Yaskawa INFORM job: OK_R2_O8B-O21B(90,0)_KMOK_HARDOX.JBI

/JOB
//NAME OK_R2_O8B-O21B(90,0)_KMOK_HARDOX
///FOLDERNAME X4
//POS
///NPOS 686,686,686,29,0,0
///TOOL 0
///POSTYPE PULSE
///PULSE
C00000=-91699,-114837,-126172,5297,65572,69852
C00001=-92194,-112793,-113721,5907,59024,69345
C00002=-143897,-89142,-104886,30363,76848,53183
C00003=-141756,-87617,-100734,29753,74573,53385
C00004=-141756,-87858,-100091,29820,74119,53263
C00005=-141756,-87802,-100249,29804,74230,53293
C00006=-141244,-84255,-98746,29497,74846,53651
C00007=-141653,-86886,-101326,29626,75189,53586
C00008=-110766,-103587,-109768,16030,63754,62789
C00009=-110766,-104046,-107477,16255,62170,62558
C00010=-110766,-104165,-106515,16351,61543,62463
C00011=-110766,-104147,-106683,16334,61651,62479
C00012=-111036,-99665,-105018,16294,62933,62564
C00013=-110753,-104252,-107692,16244,62194,62563
C00014=-67116,-81864,-100907,-8307,67410,78303
C00015=-67696,-81353,-98479,-8065,66136,78195
C00016=-67696,-81727,-97702,-8106,65471,78242
C00017=-67696,-81654,-97861,-8098,65606,78232
C00018=-68924,-78441,-96430,-7380,66259,77758
C00019=-67562,-81507,-99004,-8124,66390,78224
C00020=-94591,-107711,-114910,7081,62535,68652
C00021=-75177,-96078,-118139,30635,103857,-57240
C00022=-71016,-101172,-117038,29652,99603,-56842
C00023=-69320,-102842,-116458,29300,97976,-56637
C00024=-65815,-114376,-118551,28520,92729,-56653
C00025=-65815,-114603,-117718,28482,92175,-56787
C00026=-65333,-115185,-120736,28492,93393,-56311
C00027=-69320,-102842,-116458,29300,97976,-56637
C00028=-95175,-93300,-89498,59989,102155,-86131
C00029=-94783,-95327,-90301,59871,101628,-86283
C00030=-95175,-93300,-89498,59989,102155,-86131
C00031=-95403,-90904,-93442,60883,104178,-84663
C00032=-96846,-88575,-93381,61258,105655,-84430
C00033=-100267,-82342,-92970,62384,109223,-83757
C00034=-98853,-105972,-123361,35115,85568,-62201
C00035=-123874,-116503,-132949,35316,93358,-57662
C00036=-98784,-130821,-129289,12660,72810,-27269
C00037=-95442,-119682,-123188,11300,74256,-25961
C00038=-89918,-115832,-119261,9213,73142,-24151
C00039=-89918,-116068,-118310,9245,72445,-24204
C00040=-89918,-115832,-119261,9213,73142,-24151
C00041=-86534,-112000,-117975,7848,73961,-22933
C00042=-89918,-115832,-119261,9213,73142,-24151
C00043=-91545,-105966,-115876,9715,76271,-24462
C00044=-89918,-115832,-119261,9213,73142,-24151
C00045=-100559,-101270,-121421,12879,83175,-26784
C00046=-103898,-109015,-126857,14089,83070,-27872
C00047=-112603,-104533,-117877,29713,115926,-66306
C00048=-112603,-104533,-117877,29713,115926,-66306
C00049=-102787,-102282,-117268,28859,121596,-74546
C00050=-102787,-103288,-115881,28417,120387,-74903
C00051=-102787,-102191,-117377,28898,121696,-74514
C00052=-102247,-107992,-119426,28435,120002,-74778
C00053=-104853,-110239,-121572,27980,116786,-76632
C00054=-123177,-144145,-129947,26642,102859,-76425
C00055=-123829,-162749,-132848,26863,92935,-75206
C00056=-121638,-162916,-132889,27033,92171,-74551
C00057=-123829,-165003,-135169,26874,93176,-75150
C00058=-112500,-101779,-108680,28673,112161,-67324
C00059=-131997,-56357,-109229,-4920,90907,-66095
C00060=-147842,-82951,-112210,-34984,98309,-69155
C00061=-149737,-87239,-109966,-34223,94635,-68708
C00062=-151378,-90687,-107740,-33690,91394,-68340
C00063=-151378,-91074,-107136,-33673,90915,-68196
C00064=-151378,-90687,-107740,-33690,91394,-68340
C00065=-145558,-100693,-110774,-34812,90892,-65938
C00066=-145748,-102567,-109629,-34742,89434,-65557
C00067=-146398,-106855,-111180,-34614,88141,-65411
C00068=-145748,-102567,-109629,-34742,89434,-65557
C00069=-144942,-96836,-108242,-34942,91483,-65883
C00070=-124830,-105124,-96789,-55472,88700,-57654
C00071=-126521,-104925,-96716,-55344,87736,-58010
C00072=-123249,-105523,-98221,-55595,90026,-57599
C00073=-144949,-101354,-110618,-34915,90771,-65662
C00074=-150499,-88658,-108954,-33966,93222,-68562
C00075=-149737,-87239,-109966,-34223,94635,-68708
C00076=-147842,-82951,-112210,-34984,98309,-69155
C00077=-134744,-82461,-113999,-23220,99839,-19223
C00078=-107178,-113461,-99894,-5964,101445,70182
C00079=-116777,-120475,-92303,-7084,92443,67341
C00080=-117649,-121004,-89231,-7177,90217,67172
C00081=-117541,-124461,-90223,-7160,89070,67274
C00082=-117649,-121004,-89231,-7177,90217,67172
C00083=-121247,-121045,-89244,-7619,89875,65972
C00084=-117649,-121004,-89231,-7177,90217,67172
C00085=-120454,-123758,-93756,-7530,91322,66155
C00086=-131821,-147240,-100571,-7170,74455,63187
C00087=-132564,-146887,-99168,-7097,73320,62988
C00088=-132564,-147261,-99594,-7095,73390,62984
C00089=-116129,-123152,-95240,-7006,92928,67534
C00090=-114019,-118624,-94636,-6761,95050,68140
C00091=-115483,-77500,-114184,15325,109930,22258
C00092=-107117,-124945,-135933,-21570,97656,8797
C00093=-118143,-111392,-129277,-15030,88270,-9704
C00094=-118164,-109444,-128626,-15025,88847,-9780
C00095=-118164,-110450,-128026,-15024,87989,-9675
C00096=-118164,-110074,-128260,-15024,88315,-9716
C00097=-118257,-101380,-125250,-15013,90827,-10051
C00098=-118164,-108155,-129289,-15031,89881,-9907
C00099=-110085,-126828,-135239,-17345,85673,-6704
C00100=-92891,-111374,-130366,-26323,94899,34453
C00101=-97190,-111538,-124535,-25207,90331,33950
C00102=-98877,-113015,-125031,-24804,89436,33545
C00103=-97190,-111538,-124535,-25207,90331,33950
C00104=-97263,-106439,-128356,-25089,94874,32878
C00105=-81189,-95371,-128319,620,93628,-17487
C00106=-93710,-100817,-120600,-17770,81443,-35553
C00107=-93248,-94915,-114871,-17964,81066,-35345
C00108=-93496,-90946,-110472,-17900,80379,-35326
C00109=-93496,-91762,-109449,-17950,79378,-35179
C00110=-93496,-91644,-109606,-17943,79529,-35199
C00111=-94018,-88323,-108262,-17704,80263,-35482
C00112=-93496,-90946,-110472,-17900,80379,-35326
C00113=-94462,-94397,-113311,-17534,80159,-35616
C00114=-94975,-100261,-119034,-17317,80544,-35841
C00115=-122852,-136172,-128581,30503,68555,23673
C00116=-143305,-96642,-110194,35986,83923,20153
C00117=-143305,-96740,-110018,35993,83793,20110
C00118=-143305,-97404,-108670,36055,82835,19796
C00119=-143221,-96691,-108564,36013,83047,19900
C00120=-142576,-91782,-106634,35760,83882,20426
C00121=-143221,-96196,-109551,35968,83751,20131
C00122=-150080,-145633,-129217,38890,75983,14564
C00123=-150642,-143359,-125500,39162,75356,14082
C00124=-150642,-142275,-123303,39286,74731,13847
C00125=-150642,-142343,-123438,39278,74769,13861
C00126=-149456,-135964,-121650,38723,75947,14827
C00127=-150182,-141675,-125924,38909,76032,14540
C00128=-92946,-121634,-121424,16744,62834,34226
C00129=-86370,-109059,-114128,13073,63567,36806
C00130=-86370,-109316,-113053,13160,62794,36714
C00131=-86334,-109454,-113302,13133,62869,36736
C00132=-87103,-105692,-111971,13415,64077,36592
C00133=-86334,-109252,-114136,13065,63471,36806
C00134=-121032,-150272,-131973,30968,63431,22949
C00135=-105037,-121499,-124352,-26595,83975,43332
C00136=-119038,-120466,-118045,-23113,76809,39715
C00137=-125137,-115371,-113740,-21293,75158,37787
C00138=-125137,-115377,-112598,-21357,74498,37908
C00139=-125137,-115371,-113740,-21293,75158,37787
C00140=-125247,-119622,-115037,-21389,73833,26696
C00141=-125053,-112026,-112515,-21239,76079,26360
C00142=-125247,-119622,-115037,-21389,73833,26696
C00143=-117922,-113856,-115388,-23299,78742,39741
C00144=-113283,-118224,-119490,-24564,80311,41113
C00145=-130678,-94773,-121138,-18217,87222,14080
C00146=-167942,-138091,-131423,6732,80009,27343
C00147=-170575,-113227,-120751,7300,86397,26822
C00148=-169077,-108435,-117775,6935,86895,27340
C00149=-169077,-108900,-116810,6936,86070,27295
C00150=-169077,-108794,-117048,6936,86270,27307
C00151=-170304,-106542,-116256,7229,87038,26949
C00152=-168740,-106235,-118221,6850,88265,27525
C00153=-177701,-115390,-116622,14957,80027,1616
C00154=-176753,-112936,-115506,14676,80414,1989
C00155=-175630,-109912,-114469,14334,81107,2455
C00156=-177564,-114998,-116703,14910,80246,1690
C00157=-188009,-144692,-131667,17931,76513,-2502
C00158=-152038,-126618,-128978,-10588,85958,28176
C00159=-152038,-126618,-128978,-10588,85958,28176
C00160=-152439,-128268,-129478,-10504,85377,28090
C00161=-152439,-128687,-128060,-10515,84308,28182
C00162=-152439,-128634,-128276,-10513,84466,28168
C00163=-154807,-125417,-127295,-9971,85207,27314
C00164=-152439,-127687,-130796,-10495,86471,28000
C00165=-151563,-130369,-131601,-10695,85714,28356
C00166=-164160,-102502,-129441,9384,110509,-55546
C00167=-159433,-112173,-127809,8699,104125,-54469
C00168=-159433,-113313,-126887,8650,102984,-54550
C00169=-159433,-113125,-127052,8657,103179,-54535
C00170=-157389,-116461,-128145,8463,101945,-53942
C00171=-159433,-111320,-128398,8735,104915,-54410
C00172=-152229,-108849,-132490,7833,104970,-48789
C00173=-93963,-130535,-128792,24722,74568,-16491
C00174=-90353,-119281,-117601,23619,72522,-15568
C00175=-81815,-101184,-113078,14856,80893,-11838
C00176=-81815,-101805,-111815,14897,79832,-11967
C00177=-81815,-101566,-112336,14880,80261,-11914
C00178=-81691,-96656,-110485,14792,81580,-11713
C00179=-81815,-101566,-112336,14880,80261,-11914
C00180=-94368,-118351,-115092,25106,72713,-8195
C00181=-94368,-118242,-113051,25259,71623,-8437
C00182=-92475,-116697,-112544,24567,71499,-7736
C00183=-98770,-117080,-112671,26610,73310,-9747
C00184=-98093,-111583,-112853,26067,75742,-17780
C00185=-89023,-115119,-115343,23068,72843,-15005
C00186=-90353,-119281,-117601,23619,72522,-15568
C00187=-93963,-130636,-123354,25128,71472,-17166
C00188=-112708,-151913,-126980,52913,79334,40142
C00189=-108924,-145810,-121760,52599,77119,40924
C00190=-107448,-143466,-119685,52466,76232,41216
C00191=-107548,-140507,-116374,52568,75966,41003
C00192=-107448,-143466,-119685,52466,76232,41216
C00193=-124866,-69208,-71806,74049,113649,28483
C00194=-122400,-71971,-73000,73720,111742,28428
C00195=-124866,-69208,-71806,74049,113649,28483
C00196=-131136,-146090,-96201,76130,76771,21052
C00197=-127770,-141595,-95524,76231,74990,22221
C00198=-131136,-146090,-96201,76130,76771,21052
C00199=-112467,-159247,-111976,60211,61283,24397
C00200=-113297,-157006,-110103,60230,61789,24238
C00201=-113297,-157814,-110929,60188,61836,24279
C00202=-111416,-155256,-110381,59676,61201,25079
C00203=-114119,-159107,-112646,60032,62541,24296
C00204=-145608,-121761,-102949,57803,88894,23690
C00205=-146047,-120434,-101564,57803,89067,23542
C00206=-146481,-119084,-100092,57801,89215,23379
C00207=-146481,-119516,-101126,57808,89444,23539
C00208=-144820,-117039,-100336,57803,88864,24154
C00209=-147924,-121944,-103270,57808,90363,23296
C00210=-147924,-121944,-103270,57808,90363,23296
C00211=-137007,-126621,-110171,48785,83769,25153
C00212=-137007,-126054,-108752,48822,83378,24951
C00213=-137359,-125765,-109353,48816,83916,25050
C00214=-136478,-122214,-108258,48678,84217,25648
C00215=-137706,-129591,-111729,48871,83766,24798
C00216=-138625,-143143,-124865,48877,85014,24974
C00217=-98331,-144500,-124457,41780,63547,34680
C00218=-104311,-135778,-116637,47474,67333,33513
C00219=-104982,-134568,-114900,47757,67380,33183
C00220=-104982,-134679,-115131,47731,67438,33213
C00221=-102403,-135448,-115392,47202,65913,33778
C00222=-105649,-135232,-117175,47605,68461,33397
C00223=-103532,-169539,-136511,48991,63433,31812
C00224=-103532,-169539,-136511,48991,63433,31812
C00225=-27587,-68716,-104105,-32768,107246,55193
C00226=-44542,-60786,-93895,-29075,99837,51184
C00227=-48925,-61585,-92322,-27957,97276,50292
C00228=-49957,-62195,-92636,-27707,96857,50034
C00229=-49778,-62097,-92585,-27750,96927,50079
C00230=-49778,-62949,-91655,-27679,96029,50296
C00231=-46799,-62314,-93554,-28472,98262,50792
C00232=-32844,-112560,-114598,-30217,91594,57615
C00233=-34172,-119266,-116359,-29997,89069,57770
C00234=-36208,-121107,-116949,-29726,87845,57309
C00235=-35920,-120864,-116872,-29765,88013,57375
C00236=-35920,-120756,-115116,-29769,87119,57607
C00237=-34172,-119266,-116359,-29997,89069,57770
C00238=-34009,-88694,-103453,-33144,106213,64136
C00239=-48532,-32879,-74171,-34015,109897,57248
C00240=-43788,-34488,-76749,-34872,112199,58300
C00241=-48317,-118248,-127921,-15090,82411,66271
C00242=-90179,-134235,-132818,22872,80929,49314
C00243=-142804,-125519,-116198,76046,95508,7054
C00244=-120615,-97641,-119015,9375,90228,-9949
C00245=-120987,-96376,-113097,9471,87311,-10282
C00246=-120613,-99917,-116962,9368,87826,-10128
C00247=-121552,-104751,-117459,9639,85780,-10586
C00248=-110169,-106106,-116921,6405,83791,7848
C00249=-108950,-107035,-116988,5812,83203,8687
C00250=-101778,-109524,-117401,437,81208,17199
C00251=-92910,-108806,-115845,-6377,80483,27828
C00252=-91325,-110019,-114746,-6888,79315,28418
C00253=-89437,-130785,-128831,-4407,77618,27633
C00254=-146443,-63628,-115918,-3009,102570,37934
C00255=-146980,-83801,-122033,-27049,110301,76522
C00256=-150856,-97054,-121393,-25304,102734,76951
C00257=-152223,-100571,-121286,-24887,100651,76928
C00258=-148913,-93356,-120721,-25800,104620,77205
C00259=-150557,-96944,-122901,-25470,103711,76838
C00260=-148738,-112083,-124761,-25075,98193,78687
C00261=-146683,-119723,-126910,-25161,96417,79805
C00262=-143109,-114454,-128222,-25889,100648,80164
C00263=-140673,-104492,-128634,-26873,106197,79748
C00264=-120599,-130072,-117206,-45023,91037,77550
C00265=-120599,-129119,-114227,-44983,90071,77984
C00266=-124865,-150469,-117889,-44902,76314,77260
C00267=-120042,-124581,-111856,-45029,90980,77838
C00268=-119368,-131507,-114599,-44995,89976,78605
C00269=-124285,-150580,-117667,-44961,76466,77468
C00270=-119900,-149520,-114561,-45303,77705,79000
C00271=-119479,-146252,-112177,-45280,78069,79034
C00272=-120598,-127933,-111142,-44960,89143,78399
C00273=-120599,-129048,-114177,-44983,90075,77982
C00274=-81107,-101484,-115694,35475,102250,71567
C00275=-81237,-105179,-114207,34170,99607,71777
C00276=-82059,-102607,-116004,34567,101946,72190
C00277=-81374,-98102,-114013,34658,102588,72668
C00278=-80946,-104008,-116650,25534,103675,80963
C00279=-81739,-109308,-117836,24647,100784,82296
C00280=-83058,-108491,-117286,24741,101236,81911
C00281=-79384,-104922,-115530,34104,103743,72622
C00282=-80190,-85868,-119713,25334,110684,45677
C00283=-66991,-110384,-121517,5418,108134,-76364
C00284=-56399,-121526,-132511,11086,102541,-72269
C00285=-51570,-131189,-133992,11264,103193,-70513
C00286=-26251,-133049,-134514,-2928,99563,-63672
C00287=-67233,-108188,-115958,5335,105866,-76549
C00288=-66897,-113678,-118543,5308,104619,-76489
C00289=-40340,-135502,-134832,4529,99531,-76926
C00290=-39996,-126929,-132065,1999,104723,-72189
C00291=-40582,-118742,-129232,-2204,110819,-68387
C00292=-63906,-99170,-120419,5411,122707,-74964
C00293=-69620,-108722,-123406,2860,118643,-77498
C00294=-87784,-109018,-121307,623,118193,-84117
C00295=-84930,-119629,-129782,-1888,113436,-83486
C00296=-84729,-121080,-124653,20914,107476,-65948
C00297=-95444,-112372,-114390,31511,111945,-67927
C00298=-67316,-107916,-115567,-9495,105572,-72905
C00299=-66579,-114256,-118448,-9402,104190,-72540
C00300=-98021,-122686,-116586,31197,106837,-67491
C00301=-98017,-122619,-115764,31114,106429,-67606
C00302=-102197,-111658,-121490,32833,115802,-66493
C00303=-86428,-100957,-127747,22004,113840,-67454
C00304=-53800,-100419,-127772,-3487,91936,-72900
C00305=-55487,-108533,-124083,-2963,85444,-73257
C00306=-76650,-116115,-116137,28754,70174,-77169
C00307=-54376,-102036,-122875,-3303,88076,-72973
C00308=-53684,-106892,-125333,-3516,87122,-72731
C00309=-74308,-115452,-115917,27821,69577,-76396
C00310=-59122,-109220,-113787,21025,66918,-71130
C00311=-57844,-108351,-113482,20394,66848,-70662
C00312=-53834,-105518,-125265,-3470,87779,-72796
C00313=-58883,-114751,-131257,-1913,86567,-74352
C00314=-99205,-132197,-126076,29274,71590,12900
C00315=-100538,-139639,-126656,10769,67376,15479
C00316=-99890,-133434,-123018,10459,68226,15794
C00317=-121557,-117112,-114069,35409,80373,6489
C00318=-120930,-112739,-113965,35102,81919,7240
C00319=-105243,-128809,-121738,14815,71739,11607
C00320=-119667,-108803,-109812,34841,80971,7453
C00321=-133655,-88048,-99327,37721,90153,4837
C00322=-135782,-84357,-97373,38144,91605,4481
C00323=-120608,-113488,-111079,35194,80005,6758
C00324=-120913,-113610,-118761,34960,83981,7901
C00325=-60517,-140064,-128137,-5523,60575,30169
C00326=-76507,-136356,-126633,-15520,62258,37847
C00327=-93877,-119513,-106917,-30240,50522,43245
C00328=-93872,-118929,-104978,-30616,49748,43511
C00329=-96675,-114118,-101851,-28706,49234,42274
C00330=-91867,-119287,-104388,-32007,50022,44430
C00331=-93165,-122201,-105305,-31680,48734,44232
C00332=-96575,-112981,-98851,-29299,48158,42676
C00333=-93870,-118064,-102441,-31104,48784,43850
C00334=-93875,-120519,-110719,-29525,52112,42724
C00335=-103713,-78156,-110673,-21781,86340,9498
C00336=-103152,-115418,-123402,-33822,74617,-14862
C00337=-124928,-109292,-104782,-36694,51003,-34659
C00338=-112889,-99242,-89691,-59896,54818,-29880
C00339=-125994,-92850,-100492,-31781,60224,-38537
C00340=-127621,-94842,-100221,-31260,58610,-38740
C00341=-121155,-97272,-88940,-56496,50073,-32044
C00342=-133665,-87494,-99701,-26855,59621,-41625
C00343=-96644,-103094,-89789,-65612,59451,-20819
C00344=-121083,-121277,-109751,-27112,45366,-37764
C00345=-121016,-120747,-110300,-26892,45934,-37909
C00346=-103549,-104136,-90133,-64147,54794,-21896
C00347=-93957,-100550,-88467,-67324,63329,-21891
C00348=-159743,-124982,-101824,-32327,27989,-42293
C00349=-162261,-121311,-100710,-28180,28129,-44415
C00350=-176509,-113509,-113453,3943,47801,-53352
C00351=-120722,-118203,-110949,-26093,49137,-36520
C00352=-96719,-133488,-134181,-17465,82071,6810
C00353=-88208,-121632,-130599,-22903,100986,52847
C00354=-98918,-140805,-130229,-21227,89577,51155
C00355=-101629,-148082,-128700,-21022,84501,51062
C00356=-105953,-98261,-112767,-20869,98231,47152
C00357=-98278,-109583,-120915,-21720,99368,49630
C00358=-124341,-131813,-131636,11198,92459,-43971
C00359=-121621,-98285,-117221,11998,109073,-41436
C00360=-120746,-102076,-117837,11861,107417,-41304
C00361=-120746,-105992,-117783,11210,92936,-42669
C00362=-120747,-112603,-128286,11278,95948,-42397
C00363=-120609,-111837,-120554,26049,67413,30439
C00364=-127530,-87243,-106087,27145,76004,54708
C00365=-127898,-102267,-105837,29380,61960,54597
C00366=-120275,-109775,-109691,27025,62250,29299
C00367=-120607,-113891,-112343,27298,61925,29076
C00368=-124852,-100006,-105950,26930,63391,56220
C00369=-120420,-101837,-106812,24719,61809,57631
C00370=-119055,-102025,-106880,24011,61370,58083
C00371=-117484,-140120,-126379,-6353,63040,48502
C00372=-118425,-101447,-120931,-2723,88548,49569
C00373=-118902,-98684,-118530,-2584,88476,49421
C00374=-113028,-148150,-125976,-8643,59110,50484
C00375=-112281,-149842,-125837,-9065,58248,50850
C00376=-92052,-144569,-120194,-29364,63204,58151
C00377=-92052,-143669,-118765,-29464,62838,58255
C00378=-84683,-155167,-127701,-31711,65172,60743
C00379=-119412,-103833,-118895,-8159,86026,48306
C00380=-120645,-103801,-122240,18363,79401,46323
C00381=-120596,-133604,-113690,59811,77806,45056
C00382=-120595,-131656,-109787,60053,77075,44491
C00383=-111887,-158682,-113975,62169,55738,45421
C00384=-121130,-127010,-106775,60003,77686,44610
C00385=-122155,-131356,-109255,60198,77961,44142
C00386=-112960,-159201,-113354,62635,56094,44900
C00387=-117269,-159601,-111415,63630,58132,43433
C00388=-117569,-159775,-111136,63780,58198,43258
C00389=-120595,-130364,-107240,60219,76607,44125
C00390=-120595,-136323,-119613,59458,78987,45957
C00391=-120692,-96649,-118672,32375,84269,53596
C00392=-120600,-118120,-97579,10821,96522,62450
C00393=-120599,-116060,-93092,10778,94848,62304
C00394=-104487,-125805,-94072,2630,84980,67765
C00395=-120596,-116950,-93034,10767,94362,62263
C00396=-120597,-112553,-90859,10788,95268,62342
C00397=-105571,-126365,-94230,2579,84825,67397
C00398=-113187,-127972,-94678,2201,84500,64822
C00399=-114321,-128060,-94638,2143,84461,64439
C00400=-120599,-116103,-93113,10778,94839,62304
C00401=-120600,-118165,-97601,10821,96512,62449
C00402=-119173,-110104,-84650,-17860,100738,60179
C00403=-121454,-109687,-81979,-18272,98871,59635
C00404=-119205,-107046,-82886,-17903,101194,60099
C00405=-117500,-110311,-84228,-17454,100749,60784
C00406=-120748,-108893,-80959,-18105,98817,59897
C00407=-118360,-105961,-77958,-17548,99011,60728
C00408=-118025,-105641,-77691,-17472,99083,60836
C00409=-119269,-105795,-90384,-16222,103319,56958
C00410=-119250,-107896,-92223,-16223,103373,56958
C00411=-120631,-120794,-104165,3096,101272,-12664
C00412=-93681,-116199,-92959,21871,86687,-63192
C00413=-93682,-114281,-89064,21892,85374,-63431
C00414=-93994,-112402,-84988,21921,84020,-63792
C00415=-94896,-115380,-88949,21880,85105,-63922
C00416=-94330,-111162,-87177,21872,85957,-63561
C00417=-97211,-111244,-82023,21869,83727,-65014
C00418=-93688,-114747,-90039,16462,83105,-67478
C00419=-98020,-112989,-101813,16504,91812,-67842
C00420=-120691,-83893,-117951,31034,76795,369
C00421=-109337,-117271,-103204,33165,32410,56709
C00422=-108598,-118256,-100577,34319,30336,56092
C00423=-117079,-111264,-87799,73421,47879,44037
C00424=-120810,-118458,-98421,46795,34964,49508
C00425=-120898,-120190,-100727,46315,35380,49771
C00426=-99711,-111477,-102304,-947,36666,74602
C00427=-94382,-106967,-102468,-12697,42189,80579
C00428=-95848,-107498,-102714,-11399,41854,79888
C00429=-99681,-109355,-102836,-8004,40530,78092
C00430=-117160,-112644,-101277,9293,38000,68885
C00431=-116786,-129112,-111653,9356,35906,68838
C00432=-120602,-119646,-106124,23770,35755,64006
C00433=-120572,-164631,-130559,29498,28477,60984
C00434=-59378,-79993,-117615,20992,104349,50993
C00435=-59534,-83013,-114526,20694,101146,50372
C00436=-96077,-81408,-92413,57231,103111,43320
C00437=-79627,-66109,-85182,55504,95610,47746
C00438=-48464,-53437,-100454,18522,104822,54763
C00439=-48227,-49677,-102991,18845,108096,55363
C00440=-80679,-104141,-125686,9644,102744,40683
C00441=-118067,-125720,-131229,-18141,88550,23791
C00442=-119196,-107213,-115583,-19115,87640,23373
C00443=-121699,-105262,-112483,-19242,86972,21598
C00444=-117080,-103991,-114571,-20230,89872,22719
C00445=-116066,-108230,-114829,-20428,88214,23347
C00446=-122381,-105719,-113331,-9069,82450,8912
C00447=-126696,-108373,-114128,-6771,80419,568
C00448=-142779,-103158,-112224,8798,82570,-16248
C00449=-121247,-109622,-114889,13373,78296,-4610
C00450=-134056,-113869,-113144,-21646,71523,28395
C00451=-136867,-109744,-110142,-20577,71068,27434
C00452=-132204,-114603,-112784,-22383,71453,29101
C00453=-133799,-109730,-110978,-21650,72329,28339
C00454=-136032,-108951,-108189,-20981,70531,27843
C00455=-134059,-113755,-114816,-16878,74881,27676
C00456=-134057,-113222,-117239,-16761,76575,27439
C00457=-134085,-122795,-122723,12562,74454,-19579
C00458=-134084,-123052,-120179,12662,72796,-19752
C00459=-133873,-119304,-117433,12589,72993,-19657
C00460=-134370,-128050,-120849,12910,70736,-20076
C00461=-135935,-124649,-119997,13370,72179,-20478
C00462=-136397,-117290,-114619,14497,73201,-21549
C00463=-134086,-122982,-121548,14244,80726,-12740
C00464=-134086,-122460,-124273,14187,82615,-12522
C00465=-124281,-111431,-128342,21366,88313,4883
C00466=-101088,-90789,-125448,21651,85172,29871
C00467=-93918,-104964,-136200,23440,91622,46043
C00468=-93920,-124128,-120530,24248,73694,42461
C00469=-108956,-121485,-123239,12895,83029,39942
C00470=-107927,-162232,-128049,10374,53868,37783
C00471=-94160,-120648,-118787,24248,74418,42523
C00472=-93561,-129068,-120517,24441,71260,42079
C00473=-124294,-167626,-122785,38558,52262,22914
C00474=-137444,-156488,-111374,57751,61927,18614
C00475=-115020,-146984,-110414,53848,58947,26302
C00476=-93836,-146150,-110331,48283,47389,32108
C00477=-121737,-148346,-104693,64891,58932,23283
C00478=-104801,-149987,-105057,63967,47869,26098
C00479=-93972,-122221,-127126,23802,78331,43399
C00480=-95212,-124771,-130616,25606,80781,41793
C00481=-95212,-124771,-130616,25606,80781,41793
C00482=-95212,-124771,-130616,25606,80781,-19677
C00483=-85191,-99208,-110244,22307,78543,-16550
C00484=-85742,-100726,-104991,22819,74968,-17431
C00485=-89149,-106557,-109914,23947,75942,-18492
C00486=-123530,-75295,-101290,33091,96563,-25932
C00487=-124569,-94774,-102095,38008,80988,-30159
C00488=-124698,-95304,-97472,38342,78567,-31079
C00489=-128762,-97835,-105146,39063,83045,-31166
C00490=-66215,-117666,-119596,-4204,73122,-9588
C00491=-69871,-90584,-106325,3816,82088,-13320
C00492=-47201,-73942,-99197,-20006,93995,10785
C00493=-38626,-69356,-91924,-35532,97801,10659
C00494=-49051,-79288,-91687,-43194,92328,6604
C00495=-51006,-79528,-91797,-42852,91366,6149
C00496=-75818,-78711,-92111,-38720,85261,465
C00497=-90420,-55911,-90274,-21534,98839,11830
C00498=-83302,-63123,-101501,-23427,103509,13270
C00499=-82075,-65501,-105338,-23833,104858,13394
C00500=-96888,-120810,-128549,8566,82721,-50200
C00501=-107399,-123550,-122639,19719,77762,-53336
C00502=-105987,-126908,-125537,19297,77487,-52876
C00503=-106012,-127080,-123721,19388,76352,-53070
C00504=-99805,-77414,-105466,16976,88655,-49130
C00505=-101170,-74384,-108530,17462,92208,-49062
C00506=-110716,-78612,-119218,29200,98920,42289
C00507=-6723,-78612,-119218,29200,98920,42289
C00508=26149,-48715,-68613,-7646,64296,87864
C00509=-37227,-117034,-86146,-32359,44380,13289
C00510=-81285,-37438,-50804,-21684,56778,-30387
C00511=-80438,9168,-10717,-26405,57944,-34662
C00512=-78877,19020,-1177,-27491,57718,-33926
C00513=-78745,21063,1089,-27662,57453,-33795
C00514=-78745,21075,2041,-27832,56937,-33652
C00515=-78745,21070,1795,-27788,57069,-33689
C00516=-78800,22355,3015,-27785,56971,-33687
C00517=-78880,19396,-683,-27521,57617,-33902
C00518=-80581,13500,-4347,-26804,56376,-34308
C00519=-80587,8416,-11814,-26244,58158,-34782
C00520=-112932,28382,-4139,-2581,62718,-48966
C00521=-146242,42258,30664,20511,46292,-62528
C00522=-144329,45415,35078,19510,44794,-61921
C00523=-144704,47772,38571,20105,44001,-62295
C00524=-144704,48002,39463,20258,43596,-62390
C00525=-144704,47909,39106,20196,43758,-62352
C00526=-144309,48955,40241,19962,43508,-62207
C00527=-144794,46579,36609,19964,44584,-62204
C00528=-149300,7617,-13124,20056,55660,-61959
C00529=-110214,39149,6684,28287,96687,-48296
C00530=-93936,66202,45488,26008,82562,-45514
C00531=-94391,67020,49295,26174,80971,-46039
C00532=-94391,67246,50410,26209,80457,-46153
C00533=-94391,67082,49603,26185,80829,-46070
C00534=-95479,65713,48782,26351,80993,-46446
C00535=-95018,65028,47987,26279,80969,-46276
C00536=-95450,66206,49577,26361,80771,-46485
C00537=-95450,65446,45347,26245,82765,-46037
C00538=-89138,107882,92331,14731,87816,-82190
C00539=-89138,111019,99217,14751,85274,-82495
C00540=-89250,106756,93533,14736,86561,-82380
C00541=-89120,110339,97001,14739,86254,-82372
C00542=-90221,98751,80023,7322,86942,-46264
C00543=-89927,103084,91040,7348,82397,-46428
C00544=-89927,104680,94540,7369,81075,-46507
C00545=-89753,103519,92856,7358,81495,-46422
C00546=-89356,103608,92977,7342,81432,-46291
C00547=-89753,100048,84566,7320,84786,-46229
C00548=-90471,70344,41344,7406,96098,-45812
C00549=-106653,35973,-2775,10373,93719,-49262
C00550=-148711,-61590,-86342,17909,64527,-60132
C00551=-122925,-41472,-107688,1595,85037,-50935
C00552=-122274,54028,61959,1512,43476,-35052
C00553=-122041,57255,48823,1076,55606,-31980
C00554=-120248,71316,67884,205,51086,-31263
C00555=-120250,73921,72407,210,49640,-31267
C00556=-120250,74497,73749,211,49111,-31268
C00557=-120250,74250,73177,211,49336,-31268
C00558=-119962,76419,75825,58,48821,-31142
C00559=-120249,72234,69920,206,50305,-31267
C00560=-112329,62453,61247,-5556,54103,-20424
C00561=-112359,71771,74642,-5802,50658,-20245
C00562=-112423,63328,63484,-5579,53174,-20413
C00563=-112135,65306,64495,-5681,53586,-20316
C00564=-114102,76900,80199,-3286,51044,-19329
C00565=-115065,78556,82757,-4623,48986,-21322
C00566=-115368,69103,69060,-4259,52532,-21613
C00567=-115921,59846,55216,-3823,56258,-21985
C00568=-122274,54028,61959,1512,43476,-35052
C00569=-122925,-41472,-107688,1595,85037,-50935
C00570=-148711,-61590,-86342,17909,64527,821
C00571=-82205,52185,26528,9197,92125,77524
C00572=-80425,49732,33572,14892,75143,77168
C00573=-77799,49619,33450,14252,74688,78055
C00574=-77470,29319,12356,14028,77106,78457
C00575=-80542,29332,12371,14777,77646,77436
C00576=-80542,29183,10072,14715,78942,77593
C00577=-83444,40376,22967,15507,77364,76372
C00578=-90789,30524,28300,36708,61591,70508
C00579=-90919,34248,27781,32443,73351,74069
C00580=-90250,37957,28716,32129,74230,74603
C00581=-79524,49287,23360,8955,92284,78441
C00582=-82013,50203,28350,9162,89990,77433
C00583=-82606,66796,50707,10144,92507,77441
C00584=-81919,51967,31879,9150,88730,77372
C00585=-81934,49381,27809,9155,89894,77452
C00586=-81306,73345,58953,11716,93221,77980
C00587=-79881,50137,28283,8968,89760,78140
C00588=-80090,52101,26440,9004,91901,78222
C00589=-81396,82023,55882,32097,38956,53680
C00590=-81190,90464,69323,34749,35562,52175
C00591=-81387,100013,83485,38275,32554,50271
C00592=-81108,93968,73693,35396,34795,51817
C00593=-81117,90662,70751,35312,34890,51864
C00594=-79619,100196,83768,36674,31720,51116
C00595=-79314,90463,69327,33002,34812,53080
C00596=-79483,82000,55858,30378,38255,54553
C00597=-104233,36171,-14214,11507,86308,11753
C00598=-148711,-61590,-86342,17909,64527,-60132
C00599=-122925,-41472,-107688,1595,85037,-50935
C00600=-122274,54028,61959,1512,43476,-35052
C00601=-106492,37397,54240,2185,50844,-9950
C00602=-113507,46568,52063,21056,60301,577
C00603=-112968,55940,65611,21671,56871,98
C00604=-112656,66235,80210,22537,53356,-547
C00605=-113067,57215,68339,21946,55944,-142
C00606=-112759,58823,68838,21733,56347,74
C00607=-114859,72143,87350,23527,52696,-1663
C00608=-114945,60069,70362,22403,56644,-781
C00609=-115521,50177,56014,21714,60281,-248
C00610=-122274,54028,61959,1512,43476,-35052
C00611=-123169,-59815,-117332,1745,81551,-51041
C00612=-151982,-78435,-94523,20407,61819,-61824
C00613=-151982,-78435,-94523,20407,61819,25376
C00614=-134688,6231,-23564,20522,94268,37191
C00615=-121566,68051,47503,20391,107755,44275
C00616=-121699,66459,49653,20108,105772,43875
C00617=-120994,78473,68313,18349,104952,43951
C00618=-121400,68431,53573,20011,104381,43747
C00619=-121752,65544,48943,20095,105754,43852
C00620=-119391,75453,64951,18969,105651,44668
C00621=-119945,62314,44861,20517,106109,44598
C00622=-119825,63981,42773,20808,108088,45001
C00623=-118971,49257,27765,7041,74456,-12013
C00624=-118344,55145,37167,6948,71660,-11954
C00625=-121664,78825,65691,13749,73795,-16916
C00626=-118100,57432,39652,6887,71288,-11889
C00627=-118438,55380,38603,7006,70911,-12031
C00628=-120102,74343,60249,13375,74552,-16271
C00629=-121648,62314,45296,16341,75480,-15894
C00630=-122678,56843,36157,16407,78391,-15868
C00631=-150584,-71485,-91286,19317,62987,-61079
C00632=-123050,-50840,-112823,1671,83386,-50986
C00633=-115744,32670,26267,-2188,54498,-32210
C00634=-103599,34577,51597,1741,50803,-1907
C00635=-103485,44667,65549,1784,47401,-1921
C00636=-107915,61916,87755,11792,45049,-8610
C00637=-103440,47527,68600,1777,46992,-1909
C00638=-103682,46261,68620,1898,46335,-2027
C00639=-106641,60125,85524,12751,46171,-12114
C00640=-107897,50250,71360,13800,50416,-15577
C00641=-108788,40242,57118,13430,54084,-15447
C00642=-122274,54028,61959,1512,43476,-35052
C00643=-122925,-41472,-107688,1595,85037,-50935
C00644=-148711,-61590,-86342,17909,64527,-60132
C00645=-140484,23833,-15928,16769,94749,6864
C00646=-134656,79351,48804,15764,104925,52790
C00647=-134880,77025,49975,15594,103120,52470
C00648=-134095,98095,79314,13930,103352,52693
C00649=-134539,78416,53256,15528,101796,52420
C00650=-134970,76078,49185,15586,103137,52440
C00651=-132834,91750,71189,14288,104816,53325
C00652=-133384,71707,43609,15798,103977,53122
C00653=-133167,74106,42476,15979,105796,53445
C00654=-136631,70064,39172,19099,86104,-19657
C00655=-135438,74299,47124,18933,83255,-19683
C00656=-134720,79331,55608,18898,80594,-19843
C00657=-134970,76095,49205,18856,82809,-19586
C00658=-135406,74025,47966,18948,82624,-19770
C00659=-133469,74262,49396,18609,81460,-19260
C00660=-133939,69065,40918,18618,83988,-19040
C00661=-135132,65055,33319,18804,86739,-19035
C00662=-161684,61632,29432,16839,84695,-27584
C00663=-160372,64995,36222,16603,82080,-27487
C00664=-159643,69420,43745,16527,79671,-27561
C00665=-160448,65160,37581,16646,81374,-27609
C00666=-159857,66491,37882,16493,81734,-27354
C00667=-160958,78492,54480,16921,78071,-28247
C00668=-161774,74769,47739,16996,80384,-28212
C00669=-163061,70975,40300,17192,83167,-28272
C00670=-145516,73433,41804,7939,104800,43491
C00671=-146077,72408,44575,7815,102643,43155
C00672=-144600,83101,61245,3112,100609,51100
C00673=-146303,72040,44490,7795,102528,43069
C00674=-145797,73938,47995,7787,101309,43167
C00675=-146937,99167,81544,2811,96541,50198
C00676=-148856,87677,63203,7520,99318,41981
C00677=-148311,88144,59790,7626,101588,42310
C00678=-147556,50042,28698,13594,76773,-23660
C00679=-146399,54791,36852,13432,74072,-23552
C00680=-145796,60241,45267,13431,71657,-23607
C00681=-146486,55146,38421,13505,73324,-23667
C00682=-145946,56601,38797,13329,73737,-23427
C00683=-147986,71013,57707,14177,69976,-24604
C00684=-148727,65542,49080,14175,72522,-24569
C00685=-149878,60279,40095,14287,75466,-24633
BC00000=369159,904859,1075175
BC00001=369159,904859,1075175
BC00002=369159,904859,1075175
BC00003=369159,904859,1075175
BC00004=369159,904859,1075175
BC00005=369159,904859,1075175
BC00006=369157,904858,1075172
BC00007=369157,904858,1075172
BC00008=369159,904859,1075175
BC00009=369159,904859,1075175
BC00010=369159,904859,1075175
BC00011=369159,904859,1075175
BC00012=369159,904859,1075175
BC00013=369159,904859,1075175
BC00014=369159,904859,1075175
BC00015=369159,904859,1075175
BC00016=369159,904859,1075175
BC00017=369159,904859,1075175
BC00018=369159,904859,1075175
BC00019=369159,904859,1075175
BC00020=369159,904859,1075175
BC00021=304385,861988,1075175
BC00022=304385,861988,1075175
BC00023=304385,861988,1075175
BC00024=304385,861988,1075175
BC00025=304386,861989,1075174
BC00026=304385,861988,1075175
BC00027=304385,861988,1075175
BC00028=304385,861988,1075175
BC00029=304385,861988,1075175
BC00030=304385,861988,1075175
BC00031=304385,861988,1075175
BC00032=304385,861988,1075175
BC00033=304385,861988,1075175
BC00034=288328,899546,1075175
BC00035=281959,914244,1075175
BC00036=267248,948197,1075175
BC00037=267248,948197,1075175
BC00038=267248,948197,1075175
BC00039=267248,948197,1075175
BC00040=267248,948197,1075175
BC00041=267248,948197,1075175
BC00042=267248,948197,1075175
BC00043=267248,948197,1075175
BC00044=267248,948197,1075175
BC00045=267248,948197,1075175
BC00046=267248,948197,1075175
BC00047=235649,997683,1075175
BC00048=251913,985299,1058564
BC00049=252597,998097,1058564
BC00050=252597,998097,1058564
BC00051=252597,998097,1058564
BC00052=252597,998097,1058564
BC00053=252597,998097,1058564
BC00054=252597,998097,1058564
BC00055=252597,998097,1058564
BC00056=252597,998097,1058564
BC00057=252597,998097,1058564
BC00058=235649,940542,1075175
BC00059=303446,850180,1075175
BC00060=349702,928733,1075175
BC00061=349702,928733,1075175
BC00062=349702,928733,1075175
BC00063=349702,928733,1075175
BC00064=349702,928733,1075175
BC00065=349702,928733,1075175
BC00066=349702,928733,1075175
BC00067=349702,928733,1075175
BC00068=349702,928733,1075175
BC00069=349702,928733,1075175
BC00070=349702,928733,1075175
BC00071=349702,928733,1075175
BC00072=349702,928733,1075175
BC00073=349702,928733,1075175
BC00074=349702,928733,1075175
BC00075=349702,928733,1075175
BC00076=349702,928733,1075175
BC00077=320410,863866,1075195
BC00078=271066,805633,1075229
BC00079=271066,805633,1075229
BC00080=271067,805633,1075225
BC00081=271067,805633,1075225
BC00082=271067,805633,1075225
BC00083=271067,805633,1075225
BC00084=271067,805633,1075225
BC00085=271067,805633,1075225
BC00086=271067,805633,1075225
BC00087=271067,805633,1075225
BC00088=271067,805633,1075225
BC00089=271066,805633,1075229
BC00090=271066,805633,1075229
BC00091=239808,855616,1075200
BC00092=370689,868369,1037248
BC00093=370689,847709,1005398
BC00094=370689,847709,1005398
BC00095=370689,847709,1005398
BC00096=370689,847709,1005398
BC00097=370689,847709,1005398
BC00098=370689,847709,1005398
BC00099=370689,847709,1005398
BC00100=370689,847709,1005398
BC00101=370689,847709,1005398
BC00102=370689,847709,1005398
BC00103=370689,847709,1005398
BC00104=370176,847949,1005625
BC00105=209845,928951,1075175
BC00106=213435,937105,1075175
BC00107=213435,937105,1075175
BC00108=213435,937105,1075175
BC00109=213435,937105,1075175
BC00110=213435,937105,1075175
BC00111=213435,937105,1075175
BC00112=213435,937105,1075175
BC00113=213435,937105,1075175
BC00114=213435,937105,1075175
BC00115=89262,965988,1075175
BC00116=89262,965988,1075175
BC00117=89262,965988,1075175
BC00118=89262,965988,1075175
BC00119=89262,965988,1075175
BC00120=89262,965988,1075175
BC00121=89262,965988,1075175
BC00122=12098,1002726,1075175
BC00123=12098,1002726,1075175
BC00124=12098,1002726,1075175
BC00125=12098,1002726,1075175
BC00126=12098,1002726,1075175
BC00127=12098,1002726,1075175
BC00128=89262,965988,1075175
BC00129=89262,965988,1075175
BC00130=89262,965988,1075175
BC00131=89262,965988,1075175
BC00132=89262,965988,1075175
BC00133=89262,965988,1075175
BC00134=89262,965988,1075175
BC00135=154813,958953,1075175
BC00136=154813,958953,1075175
BC00137=154813,958953,1075175
BC00138=154813,958953,1075175
BC00139=154813,958953,1075175
BC00140=154813,958953,1075175
BC00141=154813,958953,1075175
BC00142=154813,958953,1075175
BC00143=154813,958953,1075175
BC00144=154813,958953,1075175
BC00145=146057,935891,1075175
BC00146=134994,970815,1075175
BC00147=129987,970815,1075175
BC00148=129987,970815,1075175
BC00149=129987,970815,1075175
BC00150=129987,970815,1075175
BC00151=129987,970815,1075175
BC00152=129987,970815,1075175
BC00153=129987,970815,1075175
BC00154=129987,970815,1075175
BC00155=129987,970815,1075175
BC00156=129987,970815,1075175
BC00157=129987,970815,1075175
BC00158=129987,916217,1075175
BC00159=123679,913945,1045824
BC00160=122653,913497,1036955
BC00161=122653,913497,1036955
BC00162=122653,913497,1036955
BC00163=122653,913497,1036955
BC00164=122653,913497,1036955
BC00165=122653,913497,1036955
BC00166=122653,913497,1036955
BC00167=122653,913497,1036955
BC00168=122653,913497,1036955
BC00169=122653,913497,1036955
BC00170=122653,913497,1036955
BC00171=122653,913497,1036955
BC00172=124654,917062,1041916
BC00173=141173,928857,1075175
BC00174=141173,928857,1075175
BC00175=141173,928857,1075175
BC00176=141173,928857,1075175
BC00177=141173,928857,1075175
BC00178=141173,928857,1075175
BC00179=141173,928857,1075175
BC00180=141173,928857,1075172
BC00181=141173,928857,1075172
BC00182=141173,928857,1075172
BC00183=141173,928857,1075172
BC00184=141173,928857,1075175
BC00185=141173,928857,1075175
BC00186=141173,928857,1075175
BC00187=141173,928857,1075175
BC00188=344314,843472,1075175
BC00189=344314,843472,1075175
BC00190=344314,843472,1075175
BC00191=344314,843472,1075175
BC00192=344314,843472,1075175
BC00193=344314,843472,1075175
BC00194=344314,843472,1075175
BC00195=344314,843472,1075175
BC00196=344314,843472,1075175
BC00197=344314,843472,1075175
BC00198=344314,843472,1075175
BC00199=344314,843472,1075175
BC00200=344314,843472,1075175
BC00201=344314,843472,1075175
BC00202=344314,843472,1075175
BC00203=344314,843472,1075175
BC00204=344314,843472,1075175
BC00205=344314,843472,1075175
BC00206=344314,843472,1075175
BC00207=344314,843472,1075175
BC00208=344314,843472,1075175
BC00209=344314,843472,1075175
BC00210=305706,865456,1075175
BC00211=305706,865456,1075175
BC00212=305706,865456,1075175
BC00213=305706,865456,1075175
BC00214=305706,865456,1075175
BC00215=305706,865456,1075175
BC00216=305706,865456,1075175
BC00217=305706,865456,1075175
BC00218=305706,865456,1075175
BC00219=305706,865456,1075175
BC00220=305706,865456,1075175
BC00221=305706,865456,1075175
BC00222=305706,865456,1075175
BC00223=305706,865456,1075175
BC00224=391470,812954,1075175
BC00225=391470,812954,1075175
BC00226=391470,812954,1075175
BC00227=391470,812954,1075175
BC00228=391470,812954,1075175
BC00229=391470,812954,1075175
BC00230=391470,812954,1075175
BC00231=391470,812954,1075175
BC00232=391470,812954,1075175
BC00233=391470,812954,1075175
BC00234=391470,812954,1075175
BC00235=391470,812954,1075175
BC00236=391470,812954,1075175
BC00237=391470,812954,1075175
BC00238=391470,812954,1075175
BC00239=391470,812954,1075175
BC00240=391470,812954,1075175
BC00241=391470,812954,1075175
BC00242=374573,821926,1075175
BC00243=283310,870385,1075175
BC00244=214104,898516,1075175
BC00245=217314,905507,1075172
BC00246=217315,905506,1075175
BC00247=217315,905506,1075175
BC00248=217314,905507,1075172
BC00249=217314,905507,1075172
BC00250=217314,905507,1075169
BC00251=217313,905506,1075165
BC00252=217313,905506,1075165
BC00253=216665,905570,1075166
BC00254=305976,892921,1058413
BC00255=324576,945435,1036622
BC00256=324576,945435,1036622
BC00257=324576,945435,1036622
BC00258=324576,945435,1036622
BC00259=324576,945435,1036622
BC00260=324576,945435,1036622
BC00261=324576,945435,1036622
BC00262=324576,945435,1036622
BC00263=324576,945435,1036622
BC00264=339845,945530,1075175
BC00265=334466,942806,1075175
BC00266=332315,941717,1075175
BC00267=332315,941717,1075175
BC00268=332315,941717,1075175
BC00269=332315,941717,1075175
BC00270=332315,941717,1075175
BC00271=332315,941717,1075175
BC00272=338985,941823,1075175
BC00273=344364,944547,1075175
BC00274=140011,971709,1075175
BC00275=141107,969202,1075175
BC00276=141107,969202,1075175
BC00277=141107,969202,1075175
BC00278=152187,967448,1075175
BC00279=151575,968028,1075168
BC00280=151575,968028,1075168
BC00281=141075,980904,1075175
BC00282=159724,952624,1075175
BC00283=246767,940584,1075175
BC00284=245611,987953,1075175
BC00285=273930,987953,1075175
BC00286=277246,987953,1075175
BC00287=245149,936290,1075175
BC00288=245149,936290,1075175
BC00289=277246,987953,1075175
BC00290=277246,987953,1075175
BC00291=277246,987953,1075175
BC00292=277246,987953,1075175
BC00293=277246,987953,1075175
BC00294=277246,987953,1075175
BC00295=277246,987953,1075175
BC00296=231278,1005925,1075175
BC00297=231278,1005925,1075175
BC00298=289916,904978,1075175
BC00299=289916,904978,1075175
BC00300=231278,1005925,1075175
BC00301=231278,1005925,1075175
BC00302=231278,1005925,1075175
BC00303=267695,954876,1075175
BC00304=343256,848956,1075175
BC00305=344111,848775,1075175
BC00306=323305,848750,1075174
BC00307=344234,848749,1075175
BC00308=344234,848749,1075175
BC00309=323305,848750,1075174
BC00310=323305,848750,1075174
BC00311=323305,848750,1075174
BC00312=363435,837893,1075175
BC00313=363435,837893,1075175
BC00314=263793,860022,1075175
BC00315=302564,856409,1075175
BC00316=302564,856409,1075175
BC00317=268362,866715,1075175
BC00318=268362,866715,1075175
BC00319=279359,869411,1075169
BC00320=264666,868789,1075172
BC00321=264666,868789,1075172
BC00322=264666,868789,1075172
BC00323=241357,879220,1075175
BC00324=238093,874439,1075175
BC00325=238093,874439,1075175
BC00326=307266,833486,1075175
BC00327=353426,806157,1075175
BC00328=349832,812205,1075175
BC00329=348395,814625,1075175
BC00330=348395,814625,1075175
BC00331=348395,814625,1075175
BC00332=348395,814625,1075175
BC00333=349830,812218,1075175
BC00334=353423,806170,1075175
BC00335=302722,852311,1075175
BC00336=251063,898158,1075175
BC00337=251513,932760,1075174
BC00338=251513,932760,1075174
BC00339=251513,932760,1075174
BC00340=251513,932760,1075174
BC00341=251513,932760,1075174
BC00342=251513,932760,1075174
BC00343=211391,936295,1075172
BC00344=211390,936295,1075175
BC00345=211390,936295,1075175
BC00346=211391,936295,1075172
BC00347=124269,953092,1075172
BC00348=124756,993792,1075171
BC00349=124757,993793,1075170
BC00350=124779,995671,1075171
BC00351=119426,951631,1075175
BC00352=61861,946704,1075175
BC00353=69081,970416,1065179
BC00354=69157,904970,1065179
BC00355=69157,904970,1065179
BC00356=69157,904970,1065179
BC00357=69157,904970,1065179
BC00358=69157,904970,1065179
BC00359=69157,904970,1065179
BC00360=69157,904970,1065179
BC00361=69157,904970,1065179
BC00362=69157,904970,1065179
BC00363=211099,924214,1075175
BC00364=211404,929674,1075175
BC00365=211404,929674,1075175
BC00366=211526,931858,1075175
BC00367=211526,931858,1075175
BC00368=211404,929674,1075175
BC00369=211404,929674,1075175
BC00370=211404,929674,1075175
BC00371=262656,958306,1075175
BC00372=262656,958306,1075175
BC00373=262656,958306,1075175
BC00374=262656,958306,1075175
BC00375=262656,958306,1075175
BC00376=262656,958306,1075175
BC00377=262656,958306,1075175
BC00378=262656,958306,1075175
BC00379=279593,953900,1075175
BC00380=226585,943995,1075175
BC00381=139884,992104,1075175
BC00382=144605,993116,1075175
BC00383=146493,993521,1075175
BC00384=146493,993521,1075175
BC00385=146493,993521,1075175
BC00386=146493,993521,1075175
BC00387=146493,993521,1075175
BC00388=146493,993521,1075175
BC00389=140501,991027,1075175
BC00390=135781,990015,1075175
BC00391=192425,821455,1075175
BC00392=235021,800063,1075175
BC00393=234310,796852,1075175
BC00394=234026,795567,1075173
BC00395=234026,795567,1075175
BC00396=234026,795567,1075175
BC00397=234026,795567,1075173
BC00398=234026,795567,1075173
BC00399=234026,795567,1075173
BC00400=225251,796867,1075175
BC00401=225962,800078,1075175
BC00402=290317,809215,1075175
BC00403=288632,807691,1075175
BC00404=288632,807691,1075175
BC00405=288632,807691,1075175
BC00406=288632,807691,1075175
BC00407=288632,807691,1075175
BC00408=288632,807691,1075175
BC00409=291540,805086,1075175
BC00410=291540,805086,1075175
BC00411=238711,802596,1075205
BC00412=160881,806447,1075229
BC00413=164341,802845,1075229
BC00414=165725,801404,1075229
BC00415=165725,801404,1075229
BC00416=165725,801404,1075229
BC00417=165725,801404,1075229
BC00418=170193,796260,1075229
BC00419=167597,799520,1075229
BC00420=251352,832808,1075197
BC00421=285546,898050,1075175
BC00422=287213,903274,1075175
BC00423=266028,924036,1075175
BC00424=287880,905363,1075175
BC00425=287880,905363,1075175
BC00426=300326,903390,1075171
BC00427=287881,905363,1075172
BC00428=287881,905363,1075172
BC00429=287881,905363,1075172
BC00430=287881,905363,1075172
BC00431=287881,905363,1075172
BC00432=279322,898119,1075175
BC00433=279322,898119,1075175
BC00434=309164,834294,1075175
BC00435=309164,834294,1075175
BC00436=309163,834294,1075169
BC00437=309163,834294,1075169
BC00438=309164,834294,1075175
BC00439=309164,834294,1075175
BC00440=289280,872551,1075175
BC00441=145510,956874,1075175
BC00442=140853,960362,1075175
BC00443=140620,963349,1075175
BC00444=140621,963349,1075175
BC00445=140621,963349,1075175
BC00446=122553,953196,1075175
BC00447=131814,957479,1075172
BC00448=131814,957479,1075172
BC00449=84307,950596,1075175
BC00450=172658,954491,1075175
BC00451=170431,955858,1075175
BC00452=170431,955858,1075175
BC00453=170431,955858,1075175
BC00454=170431,955858,1075175
BC00455=164883,956788,1075175
BC00456=170005,953412,1075175
BC00457=105840,949000,1075175
BC00458=108298,954456,1075175
BC00459=109281,956638,1075172
BC00460=109281,956638,1075175
BC00461=109281,956638,1075175
BC00462=109281,956638,1075172
BC00463=103754,965133,1075175
BC00464=101602,960026,1075175
BC00465=180709,946457,1075175
BC00466=274729,926897,1075175
BC00467=330665,949906,1075175
BC00468=330665,949906,1075175
BC00469=330665,949906,1075175
BC00470=330665,949906,1075175
BC00471=331151,951020,1075175
BC00472=331151,951020,1075175
BC00473=330665,949906,1075175
BC00474=330665,949906,1075175
BC00475=331151,951020,1075175
BC00476=331151,951020,1075175
BC00477=381341,942342,1075173
BC00478=381341,942342,1075173
BC00479=385559,940420,1075175
BC00480=385559,931129,1075175
BC00481=331412,819696,1075175
BC00482=331412,819696,1075175
BC00483=331412,819696,1075175
BC00484=331412,819696,1075175
BC00485=331412,819696,1075175
BC00486=331412,819696,1075175
BC00487=331412,819696,1075175
BC00488=331412,819696,1075175
BC00489=331412,819696,1075175
BC00490=331412,819696,1075175
BC00491=331412,819696,1075175
BC00492=331412,819696,1075175
BC00493=331412,819696,1075175
BC00494=331412,819696,1075175
BC00495=331413,819696,1075174
BC00496=331412,819696,1075175
BC00497=331412,819696,1075175
BC00498=331412,819696,1075175
BC00499=331412,819696,1075175
BC00500=331412,849744,1075175
BC00501=331412,849744,1075175
BC00502=331412,849744,1075175
BC00503=331412,849744,1075175
BC00504=331412,849744,1075175
BC00505=331412,849744,1075175
BC00506=330665,675227,1075175
BC00507=154521,675227,1075175
BC00508=204899,675805,820586
BC00509=216493,729795,345983
BC00510=221072,751118,158543
BC00511=221999,755433,120611
BC00512=221999,755433,120611
BC00513=221999,755433,120611
BC00514=221999,755433,120611
BC00515=221999,755433,120611
BC00516=221999,755433,120611
BC00517=221999,755433,120611
BC00518=221999,755433,120611
BC00519=221999,755433,120611
BC00520=277846,754328,149402
BC00521=340596,751644,187928
BC00522=340596,751644,187928
BC00523=340596,751644,187928
BC00524=340596,751644,187928
BC00525=340596,751644,187928
BC00526=340596,751644,187928
BC00527=340596,751644,187928
BC00528=340729,724343,187037
BC00529=265067,724343,187037
BC00530=265067,724343,187037
BC00531=265067,724343,187037
BC00532=265067,724343,187037
BC00533=265067,724343,187037
BC00534=265067,724343,187037
BC00535=265067,724343,187037
BC00536=265067,724343,187037
BC00537=265067,724343,187037
BC00538=265067,724343,187037
BC00539=265067,724343,187037
BC00540=265067,724343,187037
BC00541=265067,724343,187037
BC00542=265067,724343,187037
BC00543=265067,724343,187037
BC00544=265067,724343,187037
BC00545=265067,724343,187037
BC00546=265067,724343,187037
BC00547=265067,724343,187037
BC00548=265067,724343,187037
BC00549=286163,709095,186539
BC00550=340995,669462,185246
BC00551=119037,669462,185246
BC00552=118376,799600,385381
BC00553=117861,821566,271068
BC00554=117861,821566,271068
BC00555=117861,821566,271068
BC00556=117861,821566,271068
BC00557=117861,821566,271068
BC00558=117861,821566,271068
BC00559=117861,821566,271068
BC00560=101225,829246,304311
BC00561=101225,829246,304311
BC00562=101225,829246,304311
BC00563=101225,829246,304311
BC00564=101225,829246,304311
BC00565=101225,829246,304311
BC00566=101225,829246,304311
BC00567=101225,829246,304311
BC00568=118376,799600,385381
BC00569=119037,669462,185246
BC00570=340995,669462,185246
BC00571=249461,762322,239285
BC00572=249461,762322,239285
BC00573=249461,762322,239285
BC00574=249461,762322,239285
BC00575=249461,762322,239285
BC00576=249461,762322,239285
BC00577=249461,762322,239285
BC00578=249461,762322,239285
BC00579=249461,762322,239285
BC00580=249461,762322,239285
BC00581=249461,762322,239285
BC00582=249461,762322,239285
BC00583=249461,762322,239285
BC00584=249461,762322,239285
BC00585=249461,762322,239285
BC00586=249461,762322,239285
BC00587=249461,762322,239285
BC00588=249461,762322,239285
BC00589=180745,682763,53
BC00590=180745,682763,53
BC00591=180745,682763,53
BC00592=180745,682763,53
BC00593=180745,682763,53
BC00594=180745,682763,53
BC00595=180745,682763,53
BC00596=180745,682763,53
BC00597=276422,705889,79907
BC00598=340995,669462,185246
BC00599=119037,669462,185246
BC00600=118376,799600,385381
BC00601=97859,826740,456645
BC00602=111716,832703,379649
BC00603=111716,832703,379649
BC00604=111716,832703,379649
BC00605=111716,832703,379649
BC00606=111716,832703,379649
BC00607=111716,832703,379649
BC00608=111716,832703,379649
BC00609=111716,832703,379649
BC00610=118376,799600,385381
BC00611=119037,681159,185246
BC00612=340995,683050,185246
BC00613=340995,683050,185246
BC00614=321837,734481,215081
BC00615=307301,773502,237718
BC00616=307301,773502,237718
BC00617=307301,773502,237718
BC00618=307301,773502,237718
BC00619=307301,773502,237718
BC00620=307301,773502,237718
BC00621=307301,773502,237718
BC00622=307301,773502,237718
BC00623=316316,722241,216698
BC00624=316316,722241,216698
BC00625=316316,722241,216698
BC00626=316316,722241,216698
BC00627=316316,722241,216698
BC00628=316316,722241,216698
BC00629=316316,722241,216698
BC00630=316316,722241,216698
BC00631=340995,677587,185246
BC00632=119037,675767,185246
BC00633=118376,799600,385381
BC00634=143991,828935,462362
BC00635=143991,828935,462362
BC00636=143991,828935,462362
BC00637=143991,828935,462362
BC00638=143991,828935,462362
BC00639=143991,828935,462362
BC00640=143991,828935,462362
BC00641=143991,828935,462362
BC00642=118376,799600,385381
BC00643=119037,669462,185246
BC00644=340995,669462,185246
BC00645=343734,721892,172161
BC00646=345675,759031,162892
BC00647=345675,759031,162892
BC00648=345674,759030,162891
BC00649=345675,759031,162892
BC00650=345675,759031,162892
BC00651=345675,759031,162892
BC00652=345675,759031,162892
BC00653=345675,759031,162892
BC00654=345374,727195,137717
BC00655=345374,727195,137717
BC00656=345374,727195,137717
BC00657=345374,727195,137717
BC00658=345374,727195,137717
BC00659=345374,727195,137717
BC00660=345374,727195,137717
BC00661=345374,727195,137717
BC00662=372181,793520,137942
BC00663=372181,793520,137942
BC00664=372181,793520,137942
BC00665=372181,793520,137942
BC00666=372181,793520,137942
BC00667=372181,793520,137942
BC00668=372181,793520,137942
BC00669=372181,793520,137942
BC00670=371185,782801,182841
BC00671=371185,782801,182841
BC00672=371185,782801,182841
BC00673=371185,782801,182841
BC00674=371185,782801,182841
BC00675=371185,782801,182841
BC00676=371185,782801,182841
BC00677=371185,782801,182841
BC00678=366706,759934,216702
BC00679=366706,759934,216702
BC00680=366706,759934,216702
BC00681=366706,759934,216702
BC00682=366706,759934,216702
BC00683=366706,759934,216702
BC00684=366706,759934,216702
BC00685=366706,759934,216702
EC00000=798156,1112951
EC00001=798156,1112951
EC00002=798156,1112951
EC00003=798156,1112951
EC00004=798156,1112951
EC00005=798156,1112951
EC00006=798155,1112950
EC00007=798155,1112950
EC00008=798156,1112951
EC00009=798156,1112951
EC00010=798156,1112951
EC00011=798156,1112951
EC00012=798156,1112951
EC00013=798156,1112951
EC00014=798156,1112951
EC00015=798156,1112951
EC00016=798156,1112951
EC00017=798156,1112951
EC00018=798156,1112951
EC00019=798156,1112951
EC00020=798156,1112951
EC00021=798156,1112951
EC00022=798156,1112951
EC00023=798156,1112951
EC00024=798156,1112951
EC00025=798155,1112950
EC00026=798156,1112951
EC00027=798156,1112951
EC00028=798156,1112951
EC00029=798156,1112951
EC00030=798156,1112951
EC00031=798156,1112951
EC00032=798156,1112951
EC00033=798156,1112951
EC00034=798156,1112951
EC00035=798156,1112951
EC00036=798156,1112951
EC00037=798156,1112951
EC00038=798156,1112951
EC00039=798156,1112951
EC00040=798156,1112951
EC00041=798156,1112951
EC00042=798156,1112951
EC00043=798156,1112951
EC00044=798156,1112951
EC00045=798156,1112951
EC00046=798156,1112951
EC00047=798156,1112951
EC00048=798156,1112951
EC00049=798156,1112951
EC00050=798156,1112951
EC00051=798156,1112951
EC00052=798156,1112951
EC00053=798156,1112951
EC00054=798156,1112951
EC00055=798156,1112951
EC00056=798156,1112951
EC00057=798156,1112951
EC00058=975524,1112951
EC00059=975524,1112951
EC00060=975524,1112951
EC00061=975524,1112951
EC00062=975524,1112951
EC00063=975524,1112951
EC00064=975524,1112951
EC00065=975524,1112951
EC00066=975524,1112951
EC00067=975524,1112951
EC00068=975524,1112951
EC00069=975524,1112951
EC00070=975524,1112951
EC00071=975524,1112951
EC00072=975524,1112951
EC00073=975524,1112951
EC00074=975524,1112951
EC00075=975524,1112951
EC00076=975524,1112951
EC00077=975524,1112951
EC00078=975524,1112951
EC00079=975524,1112951
EC00080=975522,1112950
EC00081=975522,1112950
EC00082=975522,1112950
EC00083=975522,1112950
EC00084=975522,1112950
EC00085=975522,1112950
EC00086=975522,1112950
EC00087=975522,1112950
EC00088=975522,1112950
EC00089=975524,1112951
EC00090=975524,1112951
EC00091=879601,1112951
EC00092=798154,1112950
EC00093=798154,1112950
EC00094=798154,1112950
EC00095=798154,1112950
EC00096=798154,1112950
EC00097=798154,1112950
EC00098=798154,1112950
EC00099=798154,1112950
EC00100=798154,1112950
EC00101=798154,1112950
EC00102=798154,1112950
EC00103=798154,1112950
EC00104=798154,1112950
EC00105=798156,1112951
EC00106=798156,1112951
EC00107=798156,1112951
EC00108=798156,1112951
EC00109=798156,1112951
EC00110=798156,1112951
EC00111=798156,1112951
EC00112=798156,1112951
EC00113=798156,1112951
EC00114=798156,1112951
EC00115=798156,1112951
EC00116=798156,1112951
EC00117=798156,1112951
EC00118=798156,1112951
EC00119=798156,1112951
EC00120=798156,1112951
EC00121=798156,1112951
EC00122=798156,1112951
EC00123=798156,1112951
EC00124=798156,1112951
EC00125=798156,1112951
EC00126=798156,1112951
EC00127=798156,1112951
EC00128=798156,1112951
EC00129=798156,1112951
EC00130=798156,1112951
EC00131=798156,1112951
EC00132=798156,1112951
EC00133=798156,1112951
EC00134=798156,1112951
EC00135=798156,1112951
EC00136=798156,1112951
EC00137=798156,1112951
EC00138=798156,1112951
EC00139=798156,1112951
EC00140=798156,1112951
EC00141=798156,1112951
EC00142=798156,1112951
EC00143=798156,1112951
EC00144=798156,1112951
EC00145=798156,1112951
EC00146=798156,1112951
EC00147=798156,1112951
EC00148=798156,1112951
EC00149=798156,1112951
EC00150=798156,1112951
EC00151=798156,1112951
EC00152=798156,1112951
EC00153=798156,1112951
EC00154=798156,1112951
EC00155=798156,1112951
EC00156=798156,1112951
EC00157=798156,1112951
EC00158=798156,1112951
EC00159=798156,1112951
EC00160=798156,1112951
EC00161=798156,1112951
EC00162=798156,1112951
EC00163=798156,1112951
EC00164=798156,1112951
EC00165=798156,1112951
EC00166=798156,1112951
EC00167=798156,1112951
EC00168=798156,1112951
EC00169=798156,1112951
EC00170=798156,1112951
EC00171=798156,1112951
EC00172=798156,1112951
EC00173=798156,1112951
EC00174=798156,1112951
EC00175=798156,1112951
EC00176=798156,1112951
EC00177=798156,1112951
EC00178=798156,1112951
EC00179=798156,1112951
EC00180=798154,1112949
EC00181=798154,1112949
EC00182=798154,1112949
EC00183=798154,1112949
EC00184=798156,1112951
EC00185=798156,1112951
EC00186=798156,1112951
EC00187=798156,1112951
EC00188=798156,1112951
EC00189=798156,1112951
EC00190=798156,1112951
EC00191=798156,1112951
EC00192=798156,1112951
EC00193=798156,1112951
EC00194=798156,1112951
EC00195=798156,1112951
EC00196=798156,1112951
EC00197=798156,1112951
EC00198=798156,1112951
EC00199=798156,1112951
EC00200=798156,1112951
EC00201=798156,1112951
EC00202=798156,1112951
EC00203=798156,1112951
EC00204=798156,1112951
EC00205=798156,1112951
EC00206=798156,1112951
EC00207=798156,1112951
EC00208=798156,1112951
EC00209=798156,1112951
EC00210=798156,1112951
EC00211=798156,1112951
EC00212=798156,1112951
EC00213=798156,1112951
EC00214=798156,1112951
EC00215=798156,1112951
EC00216=798156,1112951
EC00217=798156,1112951
EC00218=798156,1112951
EC00219=798156,1112951
EC00220=798156,1112951
EC00221=798156,1112951
EC00222=798156,1112951
EC00223=798156,1112951
EC00224=798156,1112951
EC00225=798156,1112951
EC00226=798156,1112951
EC00227=798156,1112951
EC00228=798156,1112951
EC00229=798156,1112951
EC00230=798156,1112951
EC00231=798156,1112951
EC00232=798156,1112951
EC00233=798156,1112951
EC00234=798156,1112951
EC00235=798156,1112951
EC00236=798156,1112951
EC00237=798156,1112951
EC00238=798156,1112951
EC00239=798156,1112951
EC00240=798156,1112951
EC00241=798156,1112951
EC00242=798156,1112951
EC00243=798156,1112951
EC00244=798156,1112951
EC00245=798155,1112949
EC00246=798156,1112951
EC00247=798156,1112951
EC00248=798155,1112949
EC00249=798155,1112949
EC00250=798154,1112948
EC00251=798152,1112946
EC00252=798152,1112946
EC00253=798153,1112947
EC00254=875273,1112951
EC00255=975524,1112951
EC00256=975524,1112951
EC00257=975524,1112951
EC00258=975524,1112951
EC00259=975524,1112951
EC00260=975524,1112951
EC00261=975524,1112951
EC00262=975524,1112951
EC00263=975524,1112951
EC00264=975524,1112951
EC00265=975524,1112951
EC00266=975524,1112951
EC00267=975524,1112951
EC00268=975524,1112951
EC00269=975524,1112951
EC00270=975524,1112951
EC00271=975524,1112951
EC00272=975524,1112951
EC00273=975524,1112951
EC00274=975524,1112951
EC00275=975524,1112951
EC00276=975524,1112951
EC00277=975524,1112951
EC00278=975524,1112951
EC00279=975518,1112949
EC00280=975518,1112949
EC00281=975524,1112951
EC00282=975524,1112951
EC00283=975524,1112951
EC00284=798156,1112951
EC00285=798156,1112951
EC00286=798156,1112951
EC00287=975524,1112951
EC00288=975524,1112951
EC00289=798156,1112951
EC00290=798156,1112951
EC00291=798156,1112951
EC00292=798156,1112951
EC00293=798156,1112951
EC00294=798156,1112951
EC00295=798156,1112951
EC00296=798156,1112951
EC00297=798156,1112951
EC00298=975524,1112951
EC00299=975524,1112951
EC00300=798156,1112951
EC00301=798156,1112951
EC00302=798156,1112951
EC00303=798156,1112951
EC00304=798156,1112951
EC00305=798156,1112951
EC00306=798155,1112951
EC00307=798156,1112951
EC00308=798156,1112951
EC00309=798155,1112951
EC00310=798155,1112951
EC00311=798155,1112951
EC00312=798156,1112951
EC00313=798156,1112951
EC00314=798156,1112951
EC00315=798156,1112951
EC00316=798156,1112951
EC00317=798156,1112951
EC00318=798156,1112951
EC00319=798154,1112948
EC00320=798154,1112950
EC00321=798154,1112950
EC00322=798154,1112950
EC00323=798156,1112951
EC00324=798156,1112951
EC00325=798156,1112951
EC00326=798156,1112951
EC00327=798156,1112951
EC00328=798156,1112951
EC00329=798156,1112951
EC00330=798156,1112951
EC00331=798156,1112951
EC00332=798156,1112951
EC00333=798156,1112951
EC00334=798156,1112951
EC00335=798156,1112951
EC00336=798156,1112951
EC00337=798154,1112949
EC00338=798154,1112949
EC00339=798154,1112949
EC00340=798154,1112949
EC00341=798154,1112949
EC00342=798154,1112949
EC00343=798154,1112951
EC00344=798156,1112951
EC00345=798156,1112951
EC00346=798154,1112951
EC00347=798154,1112950
EC00348=798152,1112949
EC00349=798151,1112949
EC00350=798152,1112949
EC00351=798156,1112951
EC00352=798156,1112951
EC00353=798156,1112951
EC00354=798156,1112951
EC00355=798156,1112951
EC00356=798156,1112951
EC00357=798156,1112951
EC00358=798156,1112951
EC00359=798156,1112951
EC00360=798156,1112951
EC00361=798156,1112951
EC00362=798156,1112951
EC00363=798156,1112951
EC00364=798156,1112951
EC00365=798156,1112951
EC00366=798156,1112951
EC00367=798156,1112951
EC00368=798156,1112951
EC00369=798156,1112951
EC00370=798156,1112951
EC00371=798156,1112951
EC00372=798156,1112951
EC00373=798156,1112951
EC00374=798156,1112951
EC00375=798156,1112951
EC00376=798156,1112951
EC00377=798156,1112951
EC00378=798156,1112951
EC00379=798156,1112951
EC00380=798156,1112951
EC00381=798156,1112951
EC00382=798156,1112951
EC00383=798156,1112951
EC00384=798156,1112951
EC00385=798156,1112951
EC00386=798156,1112951
EC00387=798156,1112951
EC00388=798156,1112951
EC00389=798156,1112951
EC00390=798156,1112951
EC00391=898210,1112951
EC00392=975524,1112951
EC00393=975524,1112951
EC00394=975522,1112950
EC00395=975524,1112951
EC00396=975524,1112951
EC00397=975522,1112950
EC00398=975522,1112950
EC00399=975522,1112950
EC00400=975524,1112951
EC00401=975524,1112951
EC00402=975524,1112951
EC00403=975524,1112951
EC00404=975524,1112951
EC00405=975524,1112951
EC00406=975524,1112951
EC00407=975524,1112951
EC00408=975524,1112951
EC00409=975524,1112951
EC00410=975524,1112951
EC00411=975524,1112951
EC00412=975524,1112951
EC00413=975524,1112951
EC00414=975524,1112951
EC00415=975524,1112951
EC00416=975524,1112951
EC00417=975524,1112951
EC00418=975524,1112951
EC00419=975524,1112951
EC00420=868649,1112951
EC00421=798156,1112951
EC00422=798156,1112951
EC00423=798156,1112951
EC00424=798156,1112951
EC00425=798156,1112951
EC00426=798155,1112949
EC00427=798155,1112950
EC00428=798155,1112950
EC00429=798155,1112950
EC00430=798155,1112950
EC00431=798155,1112950
EC00432=798156,1112951
EC00433=798156,1112951
EC00434=798156,1112951
EC00435=798156,1112951
EC00436=798153,1112949
EC00437=798153,1112949
EC00438=798156,1112951
EC00439=798156,1112951
EC00440=798156,1112951
EC00441=798156,1112951
EC00442=798156,1112951
EC00443=798156,1112951
EC00444=798156,1112951
EC00445=798156,1112951
EC00446=798156,1112951
EC00447=798155,1112950
EC00448=798155,1112950
EC00449=798156,1112951
EC00450=798156,1112951
EC00451=798156,1112951
EC00452=798156,1112951
EC00453=798156,1112951
EC00454=798156,1112951
EC00455=798156,1112951
EC00456=798156,1112951
EC00457=798156,1112951
EC00458=798156,1112951
EC00459=798154,1112950
EC00460=798156,1112951
EC00461=798156,1112951
EC00462=798154,1112950
EC00463=798156,1112951
EC00464=798156,1112951
EC00465=798156,1112951
EC00466=798156,1112951
EC00467=798156,1112951
EC00468=798156,1112951
EC00469=798156,1112951
EC00470=798156,1112951
EC00471=798156,1112951
EC00472=798156,1112951
EC00473=798156,1112951
EC00474=798156,1112951
EC00475=798156,1112951
EC00476=798156,1112951
EC00477=798155,1112950
EC00478=798155,1112950
EC00479=798156,1112951
EC00480=798156,1112951
EC00481=798156,1112951
EC00482=798156,1112951
EC00483=798156,1112951
EC00484=798156,1112951
EC00485=798156,1112951
EC00486=798156,1112951
EC00487=798156,1112951
EC00488=798156,1112951
EC00489=798156,1112951
EC00490=798156,1112951
EC00491=798156,1112951
EC00492=798156,1112951
EC00493=798156,1112951
EC00494=798156,1112951
EC00495=798155,1112950
EC00496=798156,1112951
EC00497=798156,1112951
EC00498=798156,1112951
EC00499=798156,1112951
EC00500=798156,1112951
EC00501=798156,1112951
EC00502=798156,1112951
EC00503=798156,1112951
EC00504=798156,1112951
EC00505=798156,1112951
EC00506=798156,1112951
EC00507=798156,1112951
EC00508=798156,1112951
EC00509=798156,1112951
EC00510=798156,1112951
EC00511=798156,1112951
EC00512=798156,1112951
EC00513=798156,1112951
EC00514=798156,1112951
EC00515=798156,1112951
EC00516=798156,1112951
EC00517=798156,1112951
EC00518=798156,1112951
EC00519=798156,1112951
EC00520=798156,1112951
EC00521=798156,1112951
EC00522=798156,1112951
EC00523=798156,1112951
EC00524=798156,1112951
EC00525=798156,1112951
EC00526=798156,1112951
EC00527=798156,1112951
EC00528=798156,1112951
EC00529=798156,1112951
EC00530=798156,1112951
EC00531=798156,1112951
EC00532=798156,1112951
EC00533=798156,1112951
EC00534=798156,1112951
EC00535=798156,1112951
EC00536=798156,1112951
EC00537=798156,1112951
EC00538=798156,1112951
EC00539=798156,1112951
EC00540=798156,1112951
EC00541=798156,1112951
EC00542=798156,1112951
EC00543=798156,1112951
EC00544=798156,1112951
EC00545=798156,1112951
EC00546=798156,1112951
EC00547=798156,1112951
EC00548=798156,1112951
EC00549=798156,1112951
EC00550=798156,1112951
EC00551=798156,1112951
EC00552=798156,1112951
EC00553=798156,1112951
EC00554=798156,1112951
EC00555=798156,1112951
EC00556=798156,1112951
EC00557=798156,1112951
EC00558=798156,1112951
EC00559=798156,1112951
EC00560=798156,1112951
EC00561=798156,1112951
EC00562=798156,1112951
EC00563=798156,1112951
EC00564=798156,1112951
EC00565=798156,1112951
EC00566=798156,1112951
EC00567=798156,1112951
EC00568=798156,1112951
EC00569=798156,1112951
EC00570=798156,1112951
EC00571=798156,1112951
EC00572=798156,1112951
EC00573=798156,1112951
EC00574=798156,1112951
EC00575=798156,1112951
EC00576=798156,1112951
EC00577=798156,1112951
EC00578=798156,1112951
EC00579=798156,1112951
EC00580=798156,1112951
EC00581=798156,1112951
EC00582=798156,1112951
EC00583=798156,1112951
EC00584=798156,1112951
EC00585=798156,1112951
EC00586=798156,1112951
EC00587=798156,1112951
EC00588=798156,1112951
EC00589=798156,1112951
EC00590=798156,1112951
EC00591=798156,1112951
EC00592=798156,1112951
EC00593=798156,1112951
EC00594=798156,1112951
EC00595=798156,1112951
EC00596=798156,1112951
EC00597=798156,1112951
EC00598=798156,1112951
EC00599=798156,1112951
EC00600=798156,1112951
EC00601=798156,1112951
EC00602=798156,1112951
EC00603=798156,1112951
EC00604=798156,1112951
EC00605=798156,1112951
EC00606=798156,1112951
EC00607=798156,1112951
EC00608=798156,1112951
EC00609=798156,1112951
EC00610=798156,1112951
EC00611=798156,1112951
EC00612=798156,1112951
EC00613=798156,1112951
EC00614=798156,1112951
EC00615=798156,1112951
EC00616=798156,1112951
EC00617=798156,1112951
EC00618=798156,1112951
EC00619=798156,1112951
EC00620=798156,1112951
EC00621=798156,1112951
EC00622=798156,1112951
EC00623=798156,1112951
EC00624=798156,1112951
EC00625=798156,1112951
EC00626=798156,1112951
EC00627=798156,1112951
EC00628=798156,1112951
EC00629=798156,1112951
EC00630=798156,1112951
EC00631=798156,1112951
EC00632=798156,1112951
EC00633=798156,1112951
EC00634=798156,1112951
EC00635=798156,1112951
EC00636=798156,1112951
EC00637=798156,1112951
EC00638=798156,1112951
EC00639=798156,1112951
EC00640=798156,1112951
EC00641=798156,1112951
EC00642=798156,1112951
EC00643=798156,1112951
EC00644=798156,1112951
EC00645=798156,1112951
EC00646=798156,1112951
EC00647=798156,1112951
EC00648=798155,1112950
EC00649=798156,1112951
EC00650=798156,1112951
EC00651=798156,1112951
EC00652=798156,1112951
EC00653=798156,1112951
EC00654=798156,1112951
EC00655=798156,1112951
EC00656=798156,1112951
EC00657=798156,1112951
EC00658=798156,1112951
EC00659=798156,1112951
EC00660=798156,1112951
EC00661=798156,1112951
EC00662=798156,1112951
EC00663=798156,1112951
EC00664=798156,1112951
EC00665=798156,1112951
EC00666=798156,1112951
EC00667=798156,1112951
EC00668=798156,1112951
EC00669=798156,1112951
EC00670=798156,1112951
EC00671=798156,1112951
EC00672=798156,1112951
EC00673=798156,1112951
EC00674=798156,1112951
EC00675=798156,1112951
EC00676=798156,1112951
EC00677=798156,1112951
EC00678=798156,1112951
EC00679=798156,1112951
EC00680=798156,1112951
EC00681=798156,1112951
EC00682=798156,1112951
EC00683=798156,1112951
EC00684=798156,1112951
EC00685=798156,1112951
///POSTYPE BASE
///RECTAN
///RCONF 0,0,0,0,0,0,0,0,0,0,0,0,0,0,0,0,0,0,0,0,0,0,0,0
P00006=0.222,-3.123,-1.508,0.0000,0.0000,0.0000
P00021=-0.225,-6.128,-0.405,0.0000,0.0000,0.0000
P00022=0.222,-3.123,-1.508,0.0000,0.0000,0.0000
P00023=0.143,-0.036,0.682,0.0000,0.0000,0.0000
P00031=1.853,-0.001,-1.549,0.0000,0.0000,0.0000
P00032=1.957,0.503,-7.217,0.0000,0.0000,0.0000
///RCONF 0,0,0,0,1,0,0,0,0,0,0,0,0,0,0,0,0,0,0,0,0,0,0,0
P00033=-0.123,0.612,-5.012,0.0000,0.0000,0.0000
///RCONF 0,0,0,0,0,0,0,0,0,0,0,0,0,0,0,0,0,0,0,0,0,0,0,0
P00034=-0.304,0.773,-2.693,0.0000,0.0000,0.0000
P00035=2.817,0.591,-1.622,0.0000,0.0000,0.0000
P00036=-1.108,-0.829,1.850,0.0000,0.0000,0.0000
P00037=0.023,0.937,-2.677,0.0000,0.0000,0.0000
P00038=0.158,-1.133,-1.952,0.0000,0.0000,0.0000
P00039=0.012,-3.081,-0.106,0.0000,0.0000,0.0000
P00040=-0.030,9.648,2.467,0.0000,0.0000,0.0000
P00041=0.192,3.924,0.305,0.0000,0.0000,0.0000
P00042=-0.217,1.941,0.413,0.0000,0.0000,0.0000
P00043=-0.044,-1.937,1.197,0.0000,0.0000,0.0000
P00051=0.367,3.892,0.009,0.0000,0.0000,0.0000
P00052=0.088,2.832,-0.342,0.0000,0.0000,0.0000
P00055=-0.342,8.912,1.324,0.0000,0.0000,0.0000
P00056=0.568,-0.032,0.830,0.0000,0.0000,0.0000
P00057=0.586,-0.180,1.727,0.0000,0.0000,0.0000
P00058=0.385,-0.061,1.027,0.0000,0.0000,0.0000
P00059=0.483,-0.984,-2.888,0.0000,0.0000,0.0000
P00060=2.327,-2.514,-2.692,0.0000,0.0000,0.0000
P00061=1.575,-3.405,-0.752,0.0000,0.0000,0.0000
P00062=-0.135,-0.848,-1.706,0.0000,0.0000,0.0000
P00090=0.184,3.539,2.293,0.0000,0.0000,0.0000
P00091=-0.109,0.052,-0.075,0.0000,0.0000,0.0000
//INST
///DATE 2025/05/13 14:40
///ATTR SC,RW
///GROUP1 RB1,BS1
///GROUP2 ST1
NOP
'OK_r2_O8B-O21B(90,0)
'Path S3645
SFTOF3D
'POW POP KM
MOVJ C00000 BC00000 VJ=100.00  +MOVJ EC00000 VJ=100.00
MOVL C00001 BC00001 V=666.7  +MOVJ EC00001 VJ=100.00
MOVL C00002 BC00002 V=666.7  +MOVJ EC00002 VJ=0.78
SMOVL C00003 BC00003 V=166.7  +MOVJ EC00003
SREFP 3 C00004 BC00004  +REFP EC00004
CALL JOB:SEARCH-R1-S13D
SET P061 P006
SFTON3D P061
SMOVL C00005 BC00005 V=166.7  +MOVJ EC00005
SREFP 3 C00006 BC00006  +REFP EC00006
CALL JOB:SEARCH-R1-S13D
SET P061 P006
SFTON3D P061
SMOVL C00007 BC00007 V=166.7  +MOVJ EC00007
SFTOF3D
SMOVL C00008 BC00008 V=666.7  +MOVJ EC00008
SMOVL C00009 BC00009 V=166.7  +MOVJ EC00009
SREFP 3 C00010 BC00010  +REFP EC00010
CALL JOB:SEARCH-R1-S13D
SET P031 P006
SFTON3D P031
SMOVL C00011 BC00011 V=166.7  +MOVJ EC00011
SREFP 3 C00012 BC00012  +REFP EC00012
CALL JOB:SEARCH-R1-S13D
SET P031 P006
SFTON3D P031
SFTOF3D
SMOVL C00013 BC00013 V=166.7  +MOVJ EC00013
MOVL C00014 BC00014 V=666.7  +MOVJ EC00014 VJ=100.00
SMOVL C00015 BC00015 V=166.7  +MOVJ EC00015
SREFP 3 C00016 BC00016  +REFP EC00016
CALL JOB:SEARCH-R1-S13D
SET P051 P006
SFTON3D P051
SMOVL C00017 BC00017 V=166.7  +MOVJ EC00017
SREFP 3 C00018 BC00018  +REFP EC00018
CALL JOB:SEARCH-R1-S13D
SET P051 P006
SFTON3D P051
SMOVL C00019 BC00019 V=166.7  +MOVJ EC00019
MOVL C00020 BC00020 V=1000.0  +MOVJ EC00020 VJ=100.00
'Path S3646
SFTOF3D
MOVJ C00021 BC00021 VJ=100.00  +MOVJ EC00021 VJ=100.00
MOVL C00022 BC00022 V=666.7  +MOVJ EC00022 VJ=100.00
SMOVL C00023 BC00023 V=333.3  +MOVJ EC00023
SMOVL C00024 BC00024 V=166.7  +MOVJ EC00024
SREFP 3 C00025 BC00025  +REFP EC00025
CALL JOB:SEARCH-R1-S13D
SET P035 P006
SFTON3D P035
SMOVL C00026 BC00026 V=166.7  +MOVJ EC00026
SMOVL C00027 BC00027 V=250.0  +MOVJ EC00027
SMOVL C00028 BC00028 V=166.7  +MOVJ EC00028
SREFP 3 C00029 BC00029  +REFP EC00029
CALL JOB:SEARCH-R1-S13D
SET P035 P006
SFTON3D P035
SMOVL C00030 BC00030 V=166.7  +MOVJ EC00030
SMOVL C00031 BC00031 V=166.7  +MOVJ EC00031
MOVL C00032 BC00032 V=666.7  +MOVJ EC00032 VJ=100.00
MOVL C00033 BC00033 V=1000.0  +MOVJ EC00033 VJ=100.00
MOVJ C00034 BC00034 VJ=100.00  +MOVJ EC00034 VJ=100.00
'Path S3647
SFTOF3D
MOVJ C00035 BC00035 VJ=100.00  +MOVJ EC00035 VJ=100.00
MOVJ C00036 BC00036 VJ=100.00  +MOVJ EC00036 VJ=100.00
MOVL C00037 BC00037 V=666.7  +MOVJ EC00037 VJ=100.00
SMOVL C00038 BC00038 V=166.7  +MOVJ EC00038
SREFP 3 C00039 BC00039  +REFP EC00039
CALL JOB:SEARCH-R1-S13D
SET P032 P006
SFTON3D P032
SMOVL C00040 BC00040 V=166.7  +MOVJ EC00040
SREFP 3 C00041 BC00041  +REFP EC00041
CALL JOB:SEARCH-R1-S13D
SET P032 P006
SFTON3D P032
SMOVL C00042 BC00042 V=166.7  +MOVJ EC00042
SREFP 3 C00043 BC00043  +REFP EC00043
CALL JOB:SEARCH-R1-S13D
SET P032 P006
SFTON3D P032
SMOVL C00044 BC00044 V=166.7  +MOVJ EC00044
MOVL C00045 BC00045 V=666.7  +MOVJ EC00045 VJ=100.00
MOVL C00046 BC00046 V=1000.0  +MOVJ EC00046 VJ=100.00
'Path S3648
SFTOF3D
MOVJ C00047 BC00047 VJ=100.00  +MOVJ EC00047 VJ=100.00
MOVL C00048 BC00048 V=666.7  +MOVJ EC00048 VJ=100.00
SMOVL C00049 BC00049 V=166.7  +MOVJ EC00049
SREFP 3 C00050 BC00050  +REFP EC00050
CALL JOB:SEARCH-R1-S13D
SET P033 P006
SFTON3D P033
SMOVL C00051 BC00051 V=166.7  +MOVJ EC00051
SREFP 3 C00052 BC00052  +REFP EC00052
CALL JOB:SEARCH-R1-S13D
SET P033 P006
SFTON3D P033
SMOVL C00053 BC00053 V=166.7  +MOVJ EC00053
SMOVL C00054 BC00054 V=250.0  +MOVJ EC00054
SMOVL C00055 BC00055 V=166.7  +MOVJ EC00055
SREFP 3 C00056 BC00056  +REFP EC00056
CALL JOB:SEARCH-R1-S13D
SET P033 P006
SFTON3D P033
SMOVL C00057 BC00057 V=166.7  +MOVJ EC00057
MOVL C00058 BC00058 V=1000.0  +MOVJ EC00058 VJ=100.00
MOVJ C00059 BC00059 VJ=100.00  +MOVJ EC00059 VJ=100.00
'Path S3649
SFTOF3D
MOVJ C00060 BC00060 VJ=100.00  +MOVJ EC00060 VJ=100.00
MOVL C00061 BC00061 V=666.7  +MOVJ EC00061 VJ=100.00
SMOVL C00062 BC00062 V=166.7  +MOVJ EC00062
SREFP 3 C00063 BC00063  +REFP EC00063
CALL JOB:SEARCH-R1-S13D
SET P038 P006
SFTON3D P038
SMOVL C00064 BC00064 V=166.7  +MOVJ EC00064
SMOVL C00065 BC00065 V=250.0  +MOVJ EC00065
SMOVL C00066 BC00066 V=166.7  +MOVJ EC00066
SREFP 3 C00067 BC00067  +REFP EC00067
CALL JOB:SEARCH-R1-S13D
SET P038 P006
SFTON3D P038
SMOVL C00068 BC00068 V=166.7  +MOVJ EC00068
SMOVL C00069 BC00069 V=166.7  +MOVJ EC00069
SMOVL C00070 BC00070 V=166.7  +MOVJ EC00070
SREFP 3 C00071 BC00071  +REFP EC00071
CALL JOB:SEARCH-R1-S13D
SET P038 P006
SFTON3D P038
SMOVL C00072 BC00072 V=166.7  +MOVJ EC00072
SMOVL C00073 BC00073 V=200.0  +MOVJ EC00073
SMOVL C00074 BC00074 V=250.0  +MOVJ EC00074
MOVL C00075 BC00075 V=666.7  +MOVJ EC00075 VJ=100.00
MOVL C00076 BC00076 V=1000.0  +MOVJ EC00076 VJ=100.00
MOVJ C00077 BC00077 VJ=100.00  +MOVJ EC00077 VJ=100.00
'Path S3650
SFTOF3D
MOVJ C00078 BC00078 VJ=100.00  +MOVJ EC00078 VJ=100.00
MOVL C00079 BC00079 V=666.7  +MOVJ EC00079 VJ=100.00
SMOVL C00080 BC00080 V=166.7  +MOVJ EC00080
SREFP 3 C00081 BC00081  +REFP EC00081
CALL JOB:SEARCH-R1-S13D
SET P040 P006
SFTON3D P040
SMOVL C00082 BC00082 V=166.7  +MOVJ EC00082
SREFP 3 C00083 BC00083  +REFP EC00083
CALL JOB:SEARCH-R1-S13D
SET P040 P006
SFTON3D P040
SMOVL C00084 BC00084 V=166.7  +MOVJ EC00084
SMOVL C00085 BC00085 V=250.0  +MOVJ EC00085
SMOVL C00086 BC00086 V=166.7  +MOVJ EC00086
SREFP 3 C00087 BC00087  +REFP EC00087
CALL JOB:SEARCH-R1-S13D
SET P040 P006
SFTON3D P040
SMOVL C00088 BC00088 V=166.7  +MOVJ EC00088
MOVL C00089 BC00089 V=666.7  +MOVJ EC00089 VJ=100.00
MOVL C00090 BC00090 V=1000.0  +MOVJ EC00090 VJ=100.00
MOVJ C00091 BC00091 VJ=100.00  +MOVJ EC00091 VJ=100.00
'Path S3651
SFTOF3D
MOVJ C00092 BC00092 VJ=100.00  +MOVJ EC00092 VJ=100.00
MOVL C00093 BC00093 V=666.7  +MOVJ EC00093 VJ=100.00
SMOVL C00094 BC00094 V=166.7  +MOVJ EC00094
SREFP 3 C00095 BC00095  +REFP EC00095
CALL JOB:SEARCH-R1-S13D
SET P036 P006
SFTON3D P036
SMOVL C00096 BC00096 V=166.7  +MOVJ EC00096
SREFP 3 C00097 BC00097  +REFP EC00097
CALL JOB:SEARCH-R1-S13D
SET P036 P006
SFTON3D P036
SMOVL C00098 BC00098 V=166.7  +MOVJ EC00098
MOVJ C00099 BC00099 VJ=100.00  +MOVJ EC00099 VJ=100.00
MOVJ C00100 BC00100 VJ=100.00  +MOVJ EC00100 VJ=50.00
SMOVL C00101 BC00101 V=166.7  +MOVJ EC00101
SREFP 3 C00102 BC00102  +REFP EC00102
CALL JOB:SEARCH-R1-S13D
SET P036 P006
SFTON3D P036
SMOVL C00103 BC00103 V=166.7  +MOVJ EC00103
MOVL C00104 BC00104 V=666.7  +MOVJ EC00104 VJ=100.00
MOVJ C00105 BC00105 VJ=100.00  +MOVJ EC00105 VJ=100.00
'Path S3652
SFTOF3D
MOVJ C00106 BC00106 VJ=100.00  +MOVJ EC00106 VJ=100.00
MOVL C00107 BC00107 V=666.7  +MOVJ EC00107 VJ=100.00
SMOVL C00108 BC00108 V=166.7  +MOVJ EC00108
SREFP 3 C00109 BC00109  +REFP EC00109
CALL JOB:SEARCH-R1-S13D
SET P037 P006
SFTON3D P037
SMOVL C00110 BC00110 V=166.7  +MOVJ EC00110
SREFP 3 C00111 BC00111  +REFP EC00111
CALL JOB:SEARCH-R1-S13D
SET P037 P006
SFTON3D P037
SMOVL C00112 BC00112 V=166.7  +MOVJ EC00112
MOVL C00113 BC00113 V=666.7  +MOVJ EC00113 VJ=100.00
MOVL C00114 BC00114 V=1000.0  +MOVJ EC00114 VJ=100.00
'Path S3653
SFTOF3D
MOVJ C00115 BC00115 VJ=100.00  +MOVJ EC00115 VJ=100.00
MOVL C00116 BC00116 V=666.7  +MOVJ EC00116 VJ=100.00
SMOVL C00117 BC00117 V=166.7  +MOVJ EC00117
SREFP 3 C00118 BC00118  +REFP EC00118
CALL JOB:SEARCH-R1-S13D
SET P041 P006
SFTON3D P041
SMOVL C00119 BC00119 V=166.7  +MOVJ EC00119
SREFP 3 C00120 BC00120  +REFP EC00120
CALL JOB:SEARCH-R1-S13D
SET P041 P006
SFTON3D P041
SFTOF3D
SMOVL C00121 BC00121 V=166.7  +MOVJ EC00121
SMOVL C00122 BC00122 V=666.7  +MOVJ EC00122
SMOVL C00123 BC00123 V=166.7  +MOVJ EC00123
SREFP 3 C00124 BC00124  +REFP EC00124
CALL JOB:SEARCH-R1-S13D
SET P062 P006
SFTON3D P062
SMOVL C00125 BC00125 V=166.7  +MOVJ EC00125
SREFP 3 C00126 BC00126  +REFP EC00126
CALL JOB:SEARCH-R1-S13D
SET P062 P006
SFTON3D P062
SFTOF3D
SMOVL C00127 BC00127 V=166.7  +MOVJ EC00127
SMOVL C00128 BC00128 V=666.7  +MOVJ EC00128
SMOVL C00129 BC00129 V=166.7  +MOVJ EC00129
SREFP 3 C00130 BC00130  +REFP EC00130
CALL JOB:SEARCH-R1-S13D
SET P052 P006
SFTON3D P052
SMOVL C00131 BC00131 V=166.7  +MOVJ EC00131
SREFP 3 C00132 BC00132  +REFP EC00132
CALL JOB:SEARCH-R1-S13D
SET P052 P006
SFTON3D P052
SMOVL C00133 BC00133 V=166.7  +MOVJ EC00133
MOVL C00134 BC00134 V=1000.0  +MOVJ EC00134 VJ=100.00
'Path S3654
SFTOF3D
MOVJ C00135 BC00135 VJ=100.00  +MOVJ EC00135 VJ=100.00
MOVL C00136 BC00136 V=666.7  +MOVJ EC00136 VJ=100.00
SMOVL C00137 BC00137 V=166.7  +MOVJ EC00137
SREFP 3 C00138 BC00138  +REFP EC00138
CALL JOB:SEARCH-R1-S13D
SET P042 P006
SFTON3D P042
SMOVL C00139 BC00139 V=250.0  +MOVJ EC00139
SMOVL C00140 BC00140 V=166.7  +MOVJ EC00140
SREFP 3 C00141 BC00141  +REFP EC00141
CALL JOB:SEARCH-R1-S13D
SET P042 P006
SFTON3D P042
SMOVL C00142 BC00142 V=250.0  +MOVJ EC00142
MOVL C00143 BC00143 V=666.7  +MOVJ EC00143 VJ=100.00
MOVL C00144 BC00144 V=1000.0  +MOVJ EC00144 VJ=100.00
MOVJ C00145 BC00145 VJ=100.00  +MOVJ EC00145 VJ=100.00
'Path S3655
SFTOF3D
MOVJ C00146 BC00146 VJ=100.00  +MOVJ EC00146 VJ=100.00
MOVL C00147 BC00147 V=666.7  +MOVJ EC00147 VJ=100.00
SMOVL C00148 BC00148 V=166.7  +MOVJ EC00148
SREFP 3 C00149 BC00149  +REFP EC00149
CALL JOB:SEARCH-R1-S13D
SET P043 P006
SFTON3D P043
SMOVL C00150 BC00150 V=166.7  +MOVJ EC00150
SREFP 3 C00151 BC00151  +REFP EC00151
CALL JOB:SEARCH-R1-S13D
SET P043 P006
SFTON3D P043
SMOVL C00152 BC00152 V=166.7  +MOVJ EC00152
SMOVL C00153 BC00153 V=333.3  +MOVJ EC00153
SMOVL C00154 BC00154 V=166.7  +MOVJ EC00154
SREFP 3 C00155 BC00155  +REFP EC00155
CALL JOB:SEARCH-R1-S13D
SET P043 P006
SFTON3D P043
SFTOF3D
SMOVL C00156 BC00156 V=250.0  +MOVJ EC00156
MOVL C00157 BC00157 V=666.7  +MOVJ EC00157 VJ=100.00
MOVL C00158 BC00158 V=1000.0  +MOVJ EC00158 VJ=100.00
SMOVL C00159 BC00159 V=666.7  +MOVJ EC00159
SMOVL C00160 BC00160 V=166.7  +MOVJ EC00160
SREFP 3 C00161 BC00161  +REFP EC00161
CALL JOB:SEARCH-R1-S13D
SET P055 P006
SFTON3D P055
SMOVL C00162 BC00162 V=166.7  +MOVJ EC00162
SREFP 3 C00163 BC00163  +REFP EC00163
CALL JOB:SEARCH-R1-S13D
SET P055 P006
SFTON3D P055
SFTOF3D
SMOVL C00164 BC00164 V=166.7  +MOVJ EC00164
MOVJ C00165 BC00165 VJ=100.00  +MOVJ EC00165 VJ=100.00
MOVJ C00166 BC00166 VJ=100.00  +MOVJ EC00166 VJ=100.00
SMOVL C00167 BC00167 V=166.7  +MOVJ EC00167
SREFP 3 C00168 BC00168  +REFP EC00168
CALL JOB:SEARCH-R1-S13D
SET P056 P006
SFTON3D P056
SMOVL C00169 BC00169 V=166.7  +MOVJ EC00169
SREFP 3 C00170 BC00170  +REFP EC00170
CALL JOB:SEARCH-R1-S13D
SET P056 P006
SFTON3D P056
SMOVL C00171 BC00171 V=166.7  +MOVJ EC00171
MOVL C00172 BC00172 V=1000.0  +MOVJ EC00172 VJ=100.00
'Path S3656
SFTOF3D
MOVJ C00173 BC00173 VJ=100.00  +MOVJ EC00173 VJ=100.00
MOVL C00174 BC00174 V=666.7  +MOVJ EC00174 VJ=100.00
SMOVL C00175 BC00175 V=166.7  +MOVJ EC00175
SREFP 3 C00176 BC00176  +REFP EC00176
CALL JOB:SEARCH-R1-S13D
SET P039 P006
SFTON3D P039
SMOVL C00177 BC00177 V=166.7  +MOVJ EC00177
SREFP 3 C00178 BC00178  +REFP EC00178
CALL JOB:SEARCH-R1-S13D
SET P039 P006
SFTON3D P039
SMOVL C00179 BC00179 V=166.7  +MOVJ EC00179
SMOVL C00180 BC00180 V=333.3  +MOVJ EC00180
SMOVL C00181 BC00181 V=166.7  +MOVJ EC00181
SREFP 3 C00182 BC00182  +REFP EC00182
CALL JOB:SEARCH-R1-S13D
SET P039 P006
SFTON3D P039
SMOVL C00183 BC00183 V=166.7  +MOVJ EC00183
SMOVL C00184 BC00184 V=250.0  +MOVJ EC00184
SMOVL C00185 BC00185 V=416.7  +MOVJ EC00185
MOVL C00186 BC00186 V=666.7  +MOVJ EC00186 VJ=100.00
MOVL C00187 BC00187 V=1000.0  +MOVJ EC00187 VJ=100.00
'Path S3657
SFTOF3D
MOVJ C00188 BC00188 VJ=100.00  +MOVJ EC00188 VJ=100.00
MOVL C00189 BC00189 V=666.7  +MOVJ EC00189 VJ=100.00
SMOVL C00190 BC00190 V=166.7  +MOVJ EC00190
SREFP 3 C00191 BC00191  +REFP EC00191
CALL JOB:SEARCH-R1-S13D
SET P034 P006
SFTON3D P034
SMOVL C00192 BC00192 V=166.7  +MOVJ EC00192
SMOVL C00193 BC00193 V=166.7  +MOVJ EC00193
SREFP 3 C00194 BC00194  +REFP EC00194
CALL JOB:SEARCH-R1-S13D
SET P034 P006
SFTON3D P034
SMOVL C00195 BC00195 V=166.7  +MOVJ EC00195
SMOVL C00196 BC00196 V=166.7  +MOVJ EC00196
SREFP 3 C00197 BC00197  +REFP EC00197
CALL JOB:SEARCH-R1-S13D
SET P034 P006
SFTON3D P034
SMOVL C00198 BC00198 V=166.7  +MOVJ EC00198
SFTOF3D
SMOVL C00199 BC00199 V=166.7  +MOVJ EC00199
SREFP 3 C00200 BC00200  +REFP EC00200
CALL JOB:SEARCH-R1-S13D
SET P057 P006
SFTON3D P057
SMOVL C00201 BC00201 V=166.7  +MOVJ EC00201
SREFP 3 C00202 BC00202  +REFP EC00202
CALL JOB:SEARCH-R1-S13D
SET P057 P006
SFTON3D P057
SMOVL C00203 BC00203 V=166.7  +MOVJ EC00203
SFTOF3D
SMOVL C00204 BC00204 V=666.7  +MOVJ EC00204
SMOVL C00205 BC00205 V=166.7  +MOVJ EC00205
SREFP 3 C00206 BC00206  +REFP EC00206
CALL JOB:SEARCH-R1-S13D
SET P058 P006
SFTON3D P058
SMOVL C00207 BC00207 V=166.7  +MOVJ EC00207
SREFP 3 C00208 BC00208  +REFP EC00208
CALL JOB:SEARCH-R1-S13D
SET P058 P006
SFTON3D P058
SFTOF3D
SMOVL C00209 BC00209 V=166.7  +MOVJ EC00209
SMOVL C00210 BC00210 V=666.7  +MOVJ EC00210
SMOVL C00211 BC00211 V=166.7  +MOVJ EC00211
SREFP 3 C00212 BC00212  +REFP EC00212
CALL JOB:SEARCH-R1-S13D
SET P059 P006
SFTON3D P059
SMOVL C00213 BC00213 V=166.7  +MOVJ EC00213
SREFP 3 C00214 BC00214  +REFP EC00214
CALL JOB:SEARCH-R1-S13D
SET P059 P006
SFTON3D P059
SFTOF3D
SMOVL C00215 BC00215 V=166.7  +MOVJ EC00215
SMOVL C00216 BC00216 V=666.7  +MOVJ EC00216
SMOVL C00217 BC00217 V=500.0  +MOVJ EC00217
SMOVL C00218 BC00218 V=166.7  +MOVJ EC00218
SREFP 3 C00219 BC00219  +REFP EC00219
CALL JOB:SEARCH-R1-S13D
SET P060 P006
SFTON3D P060
SMOVL C00220 BC00220 V=166.7  +MOVJ EC00220
SREFP 3 C00221 BC00221  +REFP EC00221
CALL JOB:SEARCH-R1-S13D
SET P060 P006
SFTON3D P060
SMOVL C00222 BC00222 V=166.7  +MOVJ EC00222
SFTOF3D
MOVJ C00223 BC00223 VJ=100.00  +MOVJ EC00223 VJ=100.00
MOVJ C00224 BC00224 VJ=100.00  +MOVJ EC00224 VJ=100.00
MOVJ C00225 BC00225 VJ=100.00  +MOVJ EC00225 VJ=100.00
MOVJ C00226 BC00226 VJ=100.00  +MOVJ EC00226 VJ=100.00
SMOVL C00227 BC00227 V=166.7  +MOVJ EC00227
SREFP 3 C00228 BC00228  +REFP EC00228
CALL JOB:SEARCH-R1-S13D
SET P090 P006
SFTON3D P090
SMOVL C00229 BC00229 V=166.7  +MOVJ EC00229
SREFP 3 C00230 BC00230  +REFP EC00230
CALL JOB:SEARCH-R1-S13D
SET P090 P006
SFTON3D P090
SMOVL C00231 BC00231 V=166.7  +MOVJ EC00231
SFTOF3D
SMOVL C00232 BC00232 V=666.7  +MOVJ EC00232
SMOVL C00233 BC00233 V=166.7  +MOVJ EC00233
SREFP 3 C00234 BC00234  +REFP EC00234
CALL JOB:SEARCH-R1-S13D
SET P091 P006
SFTON3D P091
SMOVL C00235 BC00235 V=166.7  +MOVJ EC00235
SREFP 3 C00236 BC00236  +REFP EC00236
CALL JOB:SEARCH-R1-S13D
SET P091 P006
SFTON3D P091
SMOVL C00237 BC00237 V=166.7  +MOVJ EC00237
MACRO1 MJ#(0) ARGF6
SMOVL C00238 BC00238 V=166.7  +MOVJ EC00238
ARCON
SFTON3D P090
SMOVL C00239 BC00239 V=11.7  +MOVJ EC00239
ARCOF
SFTOF3D
SMOVL C00240 BC00240 V=166.7  +MOVJ EC00240
MOVJ C00241 BC00241 VJ=100.00  +MOVJ EC00241 VJ=100.00
MOVJ C00242 BC00242 VJ=100.00  +MOVJ EC00242 VJ=100.00
'
MOVJ C00243 BC00243 VJ=100.00  +MOVJ EC00243 VJ=100.00
'Path W3658
SFTOF3D
SFTON3D P039
MOVJ C00244 BC00244 VJ=100.00  +MOVJ EC00244 VJ=100.00
MACRO1 MJ#(0) ARGF14
SFTOF3D
SFTON3D P039
SMOVL C00245 BC00245 V=133.3  +MOVJ EC00245
SREFP 1 C00246 BC00246  +REFP EC00246
SREFP 2 C00247 BC00247  +REFP EC00247
MACRO1 MJ#(0) ARGF14
ARCON
SMOVL C00248 BC00248 V=10.0  +MOVJ EC00248
SMOVL C00249 BC00249 V=10.0  +MOVJ EC00249
SMOVL C00250 BC00250 V=11.7  +MOVJ EC00250
SMOVL C00251 BC00251 V=11.7  +MOVJ EC00251
SMOVL C00252 BC00252 V=11.7  +MOVJ EC00252
ARCOF
'Path W3659
SFTOF3D
MOVJ C00253 BC00253 VJ=25.00  +MOVJ EC00253 VJ=100.00
MOVJ C00254 BC00254 VJ=100.00  +MOVJ EC00254 VJ=100.00
'Path W3661
SFTOF3D
SFTON3D P038
MOVJ C00255 BC00255 VJ=100.00  +MOVJ EC00255 VJ=100.00
SMOVL C00256 BC00256 V=500.0  +MOVJ EC00256
SMOVL C00257 BC00257 V=133.3 PL=0  +MOVJ EC00257
SREFP 1 C00258 BC00258  +REFP EC00258
SREFP 2 C00259 BC00259  +REFP EC00259
ARCON
SMOVL C00260 BC00260 V=9.2  +MOVJ EC00260
SMOVL C00261 BC00261 V=9.2  +MOVJ EC00261
ARCOF
SMOVL C00262 BC00262 V=400.0  +MOVJ EC00262
SMOVL C00263 BC00263 V=1000.0  +MOVJ EC00263
SFTOF3D
'Path W3662
SFTOF3D
SFTON3D P038
MOVJ C00264 BC00264 VJ=100.00  +MOVJ EC00264 VJ=100.00
SMOVL C00265 BC00265 V=400.0  +MOVJ EC00265
SMOVL C00266 BC00266 V=133.3 PL=0  +MOVJ EC00266
SREFP 1 C00267 BC00267  +REFP EC00267
SREFP 2 C00268 BC00268  +REFP EC00268
ARCON
SMOVL C00269 BC00269 V=10.0  +MOVJ EC00269
SMOVL C00270 BC00270 V=10.0  +MOVJ EC00270
SMOVL C00271 BC00271 V=10.0  +MOVJ EC00271
ARCOF
SMOVL C00272 BC00272 V=400.0  +MOVJ EC00272
SMOVL C00273 BC00273 V=1000.0  +MOVJ EC00273
SFTOF3D
'Path W3663
SFTOF3D
SFTON3D P038
SMOVL C00274 BC00274 V=666.7  +MOVJ EC00274
SMOVL C00275 BC00275 V=100.0 PL=0  +MOVJ EC00275
SREFP 1 C00276 BC00276  +REFP EC00276
SREFP 2 C00277 BC00277  +REFP EC00277
ARCON
SMOVL C00278 BC00278 V=10.0  +MOVJ EC00278
SMOVL C00279 BC00279 V=10.0  +MOVJ EC00279
SMOVL C00280 BC00280 V=10.0  +MOVJ EC00280
ARCOF
SMOVL C00281 BC00281 V=400.0  +MOVJ EC00281
SFTOF3D
MOVJ C00282 BC00282 VJ=100.00  +MOVJ EC00282 VJ=100.00
'Path W3664
SFTOF3D
SFTON3D P033
MOVJ C00283 BC00283 VJ=100.00  +MOVJ EC00283 VJ=100.00
SMOVL C00284 BC00284 V=666.7  +MOVJ EC00284
SMOVL C00285 BC00285 V=666.7  +MOVJ EC00285
SMOVL C00286 BC00286 V=133.3 PL=0  +MOVJ EC00286
SREFP 1 C00287 BC00287  +REFP EC00287
SREFP 2 C00288 BC00288  +REFP EC00288
MACRO1 MJ#(0) ARGF14
ARCON
SMOVL C00289 BC00289 V=9.2  +MOVJ EC00289
SMOVL C00290 BC00290 V=9.2  +MOVJ EC00290
SMOVL C00291 BC00291 V=9.2  +MOVJ EC00291
SMOVL C00292 BC00292 V=9.2  +MOVJ EC00292
SMOVL C00293 BC00293 V=9.2  +MOVJ EC00293
SMOVL C00294 BC00294 V=9.2  +MOVJ EC00294
ARCOF
SMOVL C00295 BC00295 V=400.0  +MOVJ EC00295
SMOVL C00296 BC00296 V=1000.0  +MOVJ EC00296
SFTOF3D
'Path W3666
SFTOF3D
SFTON3D P033
SMOVL C00297 BC00297 V=133.3 PL=0  +MOVJ EC00297
SREFP 1 C00298 BC00298  +REFP EC00298
SREFP 2 C00299 BC00299  +REFP EC00299
MACRO1 MJ#(0) ARGF14
ARCON
SMOVL C00300 BC00300 V=10.0  +MOVJ EC00300
SMOVL C00301 BC00301 V=10.0  +MOVJ EC00301
ARCOF
SMOVL C00302 BC00302 V=400.0  +MOVJ EC00302
SFTOF3D
MOVJ C00303 BC00303 VJ=80.00  +MOVJ EC00303 VJ=50.00
'12
'Path W3667
SFTOF3D
SFTON3D P034
MOVJ C00304 BC00304 VJ=100.00  +MOVJ EC00304 VJ=100.00
SMOVL C00305 BC00305 V=666.7  +MOVJ EC00305
SFTON3D P034
SMOVL C00306 BC00306 V=133.3 PL=0  +MOVJ EC00306
SREFP 1 C00307 BC00307  +REFP EC00307
SREFP 2 C00308 BC00308  +REFP EC00308
MACRO1 MJ#(0) ARGF6
ARCON
COMM SWVON WEV#(21)
SMOVL C00309 BC00309 V=10.0  +MOVJ EC00309
SMOVL C00310 BC00310 V=10.0  +MOVJ EC00310
SMOVL C00311 BC00311 V=10.0  +MOVJ EC00311
ARCOF
SWVOF
SFTOF3D
SMOVL C00312 BC00312 V=400.0  +MOVJ EC00312
MOVJ C00313 BC00313 VJ=100.00  +MOVJ EC00313 VJ=15.00
'Path W3668
SFTOF3D
SFTON3D P036
MOVJ C00314 BC00314 VJ=100.00  +MOVJ EC00314 VJ=100.00
SMOVL C00315 BC00315 V=666.7  +MOVJ EC00315
SMOVL C00316 BC00316 V=133.3 PL=0  +MOVJ EC00316
SREFP 1 C00317 BC00317  +REFP EC00317
SREFP 2 C00318 BC00318  +REFP EC00318
MACRO1 MJ#(0) ARGF14
ARCON
SMOVL C00319 BC00319 V=9.2  +MOVJ EC00319
SMOVL C00320 BC00320 V=9.2  +MOVJ EC00320
SMOVL C00321 BC00321 V=9.2  +MOVJ EC00321
SMOVL C00322 BC00322 V=9.2  +MOVJ EC00322
ARCOF
SMOVL C00323 BC00323 V=400.0  +MOVJ EC00323
SMOVL C00324 BC00324 V=1000.0  +MOVJ EC00324
MOVJ C00325 BC00325 VJ=100.00  +MOVJ EC00325 VJ=15.00
MOVJ C00326 BC00326 VJ=100.00  +MOVJ EC00326 VJ=15.00
SFTON3D P036
MOVJ C00327 BC00327 VJ=100.00  +MOVJ EC00327 VJ=100.00
SMOVL C00328 BC00328 V=400.0  +MOVJ EC00328
SMOVL C00329 BC00329 V=133.3 PL=0  +MOVJ EC00329
SREFP 1 C00330 BC00330  +REFP EC00330
SREFP 2 C00331 BC00331  +REFP EC00331
MACRO1 MJ#(0) ARGF14
ARCON
SMOVL C00332 BC00332 V=10.0  +MOVJ EC00332
ARCOF
SMOVL C00333 BC00333 V=400.0  +MOVJ EC00333
SMOVL C00334 BC00334 V=1000.0  +MOVJ EC00334
SFTOF3D
'13
MOVJ C00335 BC00335 VJ=100.00  +MOVJ EC00335 VJ=100.00
MOVJ C00336 BC00336 VJ=100.00  +MOVJ EC00336 VJ=100.00
'Path W3671
SFTOF3D
SFTON3D P052
SMOVL C00337 BC00337 V=400.0  +MOVJ EC00337
MACRO1 MJ#(0) ARGF9
SMOVL C00338 BC00338 V=133.3 PL=0  +MOVJ EC00338
SREFP 1 C00339 BC00339  +REFP EC00339
SREFP 2 C00340 BC00340  +REFP EC00340
ARCON
COMM SWVON WEV#(10)
SMOVL C00341 BC00341 V=6.7  +MOVJ EC00341
ARCOF
SWVOF
SMOVL C00342 BC00342 V=166.7  +MOVJ EC00342
SFTON3D P052
SMOVL C00343 BC00343 V=133.3 PL=0  +MOVJ EC00343
SREFP 1 C00344 BC00344  +REFP EC00344
SREFP 2 C00345 BC00345  +REFP EC00345
MACRO1 MJ#(0) ARGF9
ARCON
COMM SWVON WEV#(10)
SMOVL C00346 BC00346 V=9.2  +MOVJ EC00346
SFTON3D P041
SMOVL C00347 BC00347 V=9.2  +MOVJ EC00347
SFTON3D P062
SMOVL C00348 BC00348 V=9.2  +MOVJ EC00348
SMOVL C00349 BC00349 V=9.2  +MOVJ EC00349
ARCOF
SWVOF
SMOVL C00350 BC00350 V=166.7  +MOVJ EC00350
SMOVL C00351 BC00351 V=400.0  +MOVJ EC00351
SFTOF3D
'14
'Path W3672
SFTOF3D
SFTON3D P043
MOVJ C00352 BC00352 VJ=100.00  +MOVJ EC00352 VJ=100.00
MOVJ C00353 BC00353 VJ=100.00  +MOVJ EC00353 VJ=100.00
SMOVL C00354 BC00354 V=1000.0  +MOVJ EC00354
SFTON3D P055
SMOVL C00355 BC00355 V=166.7  +MOVJ EC00355
ARCON
SMOVL C00356 BC00356 V=10.0  +MOVJ EC00356
ARCOF
SFTOF3D
MOVJ C00357 BC00357 VJ=50.00  +MOVJ EC00357 VJ=100.00
MOVJ C00358 BC00358 VJ=100.00  +MOVJ EC00358 VJ=50.00
SFTON3D P056
SMOVL C00359 BC00359 V=250.0  +MOVJ EC00359
SMOVL C00360 BC00360 V=133.3  +MOVJ EC00360
ARCON
SMOVL C00361 BC00361 V=10.0  +MOVJ EC00361
ARCOF
SMOVL C00362 BC00362 V=333.3  +MOVJ EC00362
SFTOF3D
'15-brak
'16
'Path W3673
SFTOF3D
SFTON3D P037
MOVJ C00363 BC00363 VJ=100.00  +MOVJ EC00363 VJ=100.00
SMOVL C00364 BC00364 V=666.7  +MOVJ EC00364
SMOVL C00365 BC00365 V=133.3 PL=0  +MOVJ EC00365
SREFP 1 C00366 BC00366  +REFP EC00366
SREFP 2 C00367 BC00367  +REFP EC00367
MACRO1 MJ#(0) ARGF14
ARCON
SMOVL C00368 BC00368 V=10.0  +MOVJ EC00368
SMOVL C00369 BC00369 V=10.0  +MOVJ EC00369
SMOVL C00370 BC00370 V=10.0  +MOVJ EC00370
ARCOF
SFTOF3D
SFTON3D P037
SMOVL C00371 BC00371 V=166.7 PL=0  +MOVJ EC00371
SREFP 1 C00372 BC00372  +REFP EC00372
SREFP 2 C00373 BC00373  +REFP EC00373
ARCON
SMOVL C00374 BC00374 V=10.0  +MOVJ EC00374
SMOVL C00375 BC00375 V=10.0  +MOVJ EC00375
ARCON
SMOVL C00376 BC00376 V=10.0  +MOVJ EC00376
SMOVL C00377 BC00377 V=10.8  +MOVJ EC00377
ARCOF
SMOVL C00378 BC00378 V=250.0  +MOVJ EC00378
SMOVL C00379 BC00379 V=400.0  +MOVJ EC00379
SFTOF3D
MOVJ C00380 BC00380 VJ=100.00  +MOVJ EC00380 VJ=100.00
'Path W3675
SFTOF3D
SFTON3D P037
MOVJ C00381 BC00381 VJ=100.00  +MOVJ EC00381 VJ=100.00
SMOVL C00382 BC00382 V=400.0  +MOVJ EC00382
SMOVL C00383 BC00383 V=166.7 PL=0  +MOVJ EC00383
SREFP 1 C00384 BC00384  +REFP EC00384
SREFP 2 C00385 BC00385  +REFP EC00385
ARCON
SMOVL C00386 BC00386 V=10.0  +MOVJ EC00386
SMOVL C00387 BC00387 V=10.0  +MOVJ EC00387
SMOVL C00388 BC00388 V=10.0  +MOVJ EC00388
ARCOF
SMOVL C00389 BC00389 V=400.0  +MOVJ EC00389
SMOVL C00390 BC00390 V=1000.0  +MOVJ EC00390
SFTOF3D
'17
MOVJ C00391 BC00391 VJ=100.00  +MOVJ EC00391 VJ=100.00
'Path W3676
SFTOF3D
SFTON3D P040
MOVJ C00392 BC00392 VJ=100.00  +MOVJ EC00392 VJ=100.00
SMOVL C00393 BC00393 V=400.0  +MOVJ EC00393
SMOVL C00394 BC00394 V=166.7 PL=0  +MOVJ EC00394
SREFP 1 C00395 BC00395  +REFP EC00395
SREFP 2 C00396 BC00396  +REFP EC00396
ARCON
SMOVL C00397 BC00397 V=10.0  +MOVJ EC00397
SMOVL C00398 BC00398 V=10.0  +MOVJ EC00398
SMOVL C00399 BC00399 V=10.0  +MOVJ EC00399
ARCOF
SMOVL C00400 BC00400 V=400.0  +MOVJ EC00400
SMOVL C00401 BC00401 V=1000.0  +MOVJ EC00401
SFTOF3D
'Path W3677
SFTOF3D
SFTON3D P040
SMOVL C00402 BC00402 V=400.0  +MOVJ EC00402
SMOVL C00403 BC00403 V=133.3 PL=0  +MOVJ EC00403
SREFP 1 C00404 BC00404  +REFP EC00404
SREFP 2 C00405 BC00405  +REFP EC00405
ARCON
SMOVL C00406 BC00406 V=10.0  +MOVJ EC00406
SMOVL C00407 BC00407 V=10.0  +MOVJ EC00407
SMOVL C00408 BC00408 V=10.0  +MOVJ EC00408
ARCOF
SMOVL C00409 BC00409 V=400.0  +MOVJ EC00409
MOVJ C00410 BC00410 VJ=100.00  +MOVJ EC00410 VJ=50.00
SFTOF3D
MOVJ C00411 BC00411 VJ=100.00  +MOVJ EC00411 VJ=100.00
'Path W3678
SFTOF3D
SFTON3D P040
SFTOF3D
MOVJ C00412 BC00412 VJ=100.00  +MOVJ EC00412 VJ=100.00
SMOVL C00413 BC00413 V=400.0  +MOVJ EC00413
SMOVL C00414 BC00414 V=133.3 PL=0  +MOVJ EC00414
SREFP 1 C00415 BC00415  +REFP EC00415
SREFP 2 C00416 BC00416  +REFP EC00416
MACRO1 MJ#(0) ARGF14
SMOVL C00417 BC00417 V=25.0  +MOVJ EC00417
ARCOF
SMOVL C00418 BC00418 V=400.0  +MOVJ EC00418
SMOVL C00419 BC00419 V=1000.0  +MOVJ EC00419
SFTOF3D
'18
MOVJ C00420 BC00420 VJ=100.00  +MOVJ EC00420 VJ=100.00
'Path W3679
SFTOF3D
SFTOF3D
SFTON3D P032
MOVJ C00421 BC00421 VJ=100.00  +MOVJ EC00421 VJ=100.00
SMOVL C00422 BC00422 V=400.0  +MOVJ EC00422
SMOVL C00423 BC00423 V=166.7  +MOVJ EC00423
SREFP 1 C00424 BC00424  +REFP EC00424
SREFP 2 C00425 BC00425  +REFP EC00425
MACRO1 MJ#(0) ARGF14
ARCON
SMOVL C00426 BC00426 V=9.2  +MOVJ EC00426
SMOVL C00427 BC00427 V=9.2  +MOVJ EC00427
SMOVL C00428 BC00428 V=9.2  +MOVJ EC00428
SMOVL C00429 BC00429 V=9.2  +MOVJ EC00429
SMOVL C00430 BC00430 V=9.2  +MOVJ EC00430
ARCOF
SMOVL C00431 BC00431 V=400.0  +MOVJ EC00431
SFTOF3D
'Path W3680
SMOVL C00432 BC00432 V=1000.0  +MOVJ EC00432
SFTOF3D
'19
MOVJ C00433 BC00433 VJ=100.00  +MOVJ EC00433 VJ=70.00
'Path W3681
SFTOF3D
SFTON3D P035
MOVJ C00434 BC00434 VJ=100.00  +MOVJ EC00434 VJ=100.00
SMOVL C00435 BC00435 V=400.0  +MOVJ EC00435
SMOVL C00436 BC00436 V=133.3 PL=0  +MOVJ EC00436
MACRO1 MJ#(0) ARGF6
ARCON
COMM SWVON WEV#(21)
SMOVL C00437 BC00437 V=9.2  +MOVJ EC00437
ARCOF
SWVOF
SMOVL C00438 BC00438 V=400.0  +MOVJ EC00438
SMOVL C00439 BC00439 V=1000.0  +MOVJ EC00439
SFTOF3D
'20
MOVJ C00440 BC00440 VJ=100.00  +MOVJ EC00440 VJ=100.00
MOVJ C00441 BC00441 VJ=100.00  +MOVJ EC00441 VJ=100.00
'Path W3682
SFTOF3D
SFTON3D P042
SMOVL C00442 BC00442 V=400.0  +MOVJ EC00442
SMOVL C00443 BC00443 V=133.3 PL=0  +MOVJ EC00443
SREFP 1 C00444 BC00444  +REFP EC00444
SREFP 2 C00445 BC00445  +REFP EC00445
MACRO1 MJ#(0) ARGF6
ARCON
SMOVL C00446 BC00446 V=7.5  +MOVJ EC00446
SMOVL C00447 BC00447 V=7.5  +MOVJ EC00447
SMOVL C00448 BC00448 V=7.5  +MOVJ EC00448
ARCOF
SMOVL C00449 BC00449 V=400.0  +MOVJ EC00449
SFTOF3D
SFTON3D P042
SMOVL C00450 BC00450 V=400.0  +MOVJ EC00450
SMOVL C00451 BC00451 V=133.3 PL=0  +MOVJ EC00451
SREFP 1 C00452 BC00452  +REFP EC00452
SREFP 2 C00453 BC00453  +REFP EC00453
MACRO1 MJ#(0) ARGF6
ARCON
SMOVL C00454 BC00454 V=10.0  +MOVJ EC00454
ARCOF
SMOVL C00455 BC00455 V=400.0  +MOVJ EC00455
SMOVL C00456 BC00456 V=1000.0  +MOVJ EC00456
SFTOF3D
'Path W3686
SFTOF3D
SFTON3D P042
MOVJ C00457 BC00457 VJ=100.00  +MOVJ EC00457 VJ=100.00
SMOVL C00458 BC00458 V=400.0  +MOVJ EC00458
SMOVL C00459 BC00459 V=166.7 PL=0  +MOVJ EC00459
SREFP 1 C00460 BC00460  +REFP EC00460
SREFP 2 C00461 BC00461  +REFP EC00461
MACRO1 MJ#(0) ARGF6
ARCON
SMOVL C00462 BC00462 V=10.0  +MOVJ EC00462
ARCOF
SMOVL C00463 BC00463 V=400.0  +MOVJ EC00463
SMOVL C00464 BC00464 V=1000.0  +MOVJ EC00464
SFTOF3D
'21
MOVJ C00465 BC00465 VJ=100.00  +MOVJ EC00465 VJ=100.00
MOVJ C00466 BC00466 VJ=100.00  +MOVJ EC00466 VJ=100.00
MOVJ C00467 BC00467 VJ=70.00  +MOVJ EC00467 VJ=70.00
'Path W3687
SFTOF3D
SFTON3D P061
SMOVL C00468 BC00468 V=833.3  +MOVJ EC00468
SMOVL C00469 BC00469 V=666.7  +MOVJ EC00469
SMOVL C00470 BC00470 V=166.7 PL=0  +MOVJ EC00470
SREFP 1 C00471 BC00471  +REFP EC00471
SREFP 2 C00472 BC00472  +REFP EC00472
MACRO1 MJ#(0) ARGF9
ARCON
SMOVL C00473 BC00473 V=10.8  +MOVJ EC00473
SMOVL C00474 BC00474 V=10.8  +MOVJ EC00474
SFTON3D P031
SMOVL C00475 BC00475 V=10.8  +MOVJ EC00475
SMOVL C00476 BC00476 V=10.8  +MOVJ EC00476
SFTON3D P051
SMOVL C00477 BC00477 V=12.5  +MOVJ EC00477
SMOVL C00478 BC00478 V=12.5  +MOVJ EC00478
ARCOF
SMOVL C00479 BC00479 V=400.0  +MOVJ EC00479
MOVJ C00480 BC00480 VJ=100.00  +MOVJ EC00480 VJ=50.00
MOVJ C00481 BC00481 VJ=100.00  +MOVJ EC00481 VJ=50.00
MACRO1 MJ#(0) ARGF14
MOVJ C00482 BC00482 VJ=100.00  +MOVJ EC00482 VJ=100.00
SFTON3D P034
SMOVL C00483 BC00483 V=166.7  +MOVJ EC00483
ARCON
SMOVL C00484 BC00484 V=10.0  +MOVJ EC00484
ARCOF
SMOVL C00485 BC00485 V=166.7  +MOVJ EC00485
SFTOF3D
SMOVL C00486 BC00486 V=333.3  +MOVJ EC00486
SFTOF3D
MACRO1 MJ#(0) ARGF9
SFTON3D P058
SMOVL C00487 BC00487 V=166.7  +MOVJ EC00487
ARCON
SMOVL C00488 BC00488 V=11.7  +MOVJ EC00488
ARCOF
SMOVL C00489 BC00489 V=333.3  +MOVJ EC00489
SFTOF3D
SMOVL C00490 BC00490 V=333.3  +MOVJ EC00490
MACRO1 MJ#(0) ARGF9
SFTON3D P057
SMOVL C00491 BC00491 V=166.7 PL=0  +MOVJ EC00491
ARCON
SMOVL C00492 BC00492 V=9.2  +MOVJ EC00492
SFTON3D P058
SMOVL C00493 BC00493 V=9.2  +MOVJ EC00493
SMOVL C00494 BC00494 V=9.2  +MOVJ EC00494
SFTON3D P059
COMM SWVON WEV#(30)
SMOVL C00495 BC00495 V=8.7  +MOVJ EC00495
SMOVL C00496 BC00496 V=8.7  +MOVJ EC00496
SMOVL C00497 BC00497 V=8.7  +MOVJ EC00497
ARCOF
SWVOF
SFTOF3D
SMOVL C00498 BC00498 V=250.0  +MOVJ EC00498
MOVJ C00499 BC00499 VJ=100.00  +MOVJ EC00499 VJ=100.00
MOVJ C00500 BC00500 VJ=100.00  +MOVJ EC00500 VJ=100.00
SFTON3D P060
SREFP 1 C00501 BC00501  +REFP EC00501
SREFP 2 C00502 BC00502  +REFP EC00502
SMOVL C00503 BC00503 V=250.0  +MOVJ EC00503
ARCON
COMM SWVON WEV#(12)
SMOVL C00504 BC00504 V=10.0  +MOVJ EC00504
ARCOF
SWVOF
SMOVL C00505 BC00505 V=250.0  +MOVJ EC00505
SFTOF3D
MOVJ C00506 BC00506 VJ=100.00  +MOVJ EC00506 VJ=100.00
MOVJ C00507 BC00507 VJ=100.00  +MOVJ EC00507 VJ=70.00
CALL JOB:CLEAN-R1_KM_3P
MOVJ C00508 BC00508 VJ=100.00  +MOVJ EC00508 VJ=100.00
'cut_wire_dol
'Path S3688
SFTOF3D
MOVJ C00509 BC00509 VJ=100.00  +MOVJ EC00509 VJ=70.00
MOVJ C00510 BC00510 VJ=100.00  +MOVJ EC00510 VJ=70.00
MOVJ C00511 BC00511 VJ=100.00  +MOVJ EC00511 VJ=100.00
MOVL C00512 BC00512 V=400.0  +MOVJ EC00512 VJ=100.00
SMOVL C00513 BC00513 V=100.0  +MOVJ EC00513
SREFP 3 C00514 BC00514  +REFP EC00514
CALL JOB:SEARCH-R1-S13D
SET P023 P006
SFTON3D P023
SMOVL C00515 BC00515 V=100.0  +MOVJ EC00515
SREFP 3 C00516 BC00516  +REFP EC00516
CALL JOB:SEARCH-R1-S13D
SET P023 P006
SFTON3D P023
SMOVL C00517 BC00517 V=100.0  +MOVJ EC00517
MOVL C00518 BC00518 V=400.0  +MOVJ EC00518 VJ=100.00
